LIN {X 0,Y 418.321,Z 60.369,A -85,B 0,C 180,E1 -10243.405,E2 -10243.405} C_VEL
LIN {X 0,Y 418.35,Z 60.367,A -85,B 0,C 180,E1 -10246.999,E2 -10246.999} C_VEL
LIN {X 0,Y 418.344,Z 60.377,A -85,B 0,C 180,E1 -10250.329,E2 -10250.329} C_VEL
LIN {X 0,Y 418.492,Z 60.345,A -85,B 0,C 180,E1 -10253.249,E2 -10253.249} C_VEL
LIN {X 0,Y 418.34,Z 60.372,A -85,B 0,C 180,E1 -10255.181,E2 -10255.181} C_VEL
LIN {X 0,Y 418.544,Z 60.343,A -85,B 0,C 180,E1 -10258.075,E2 -10258.075} C_VEL
LIN {X 0,Y 418.675,Z 60.334,A -85,B 0,C 180,E1 -10260,E2 -10260} C_VEL
LIN {X 0,Y 418.503,Z 60.349,A -85,B 0,C 180,E1 -10262.888,E2 -10262.888} C_VEL
LIN {X 0,Y 418.47,Z 60.356,A -85,B 0,C 180,E1 -10266.618,E2 -10266.618} C_VEL
LIN {X 0,Y 418.342,Z 60.372,A -85,B 0,C 180,E1 -10269.671,E2 -10269.671} C_VEL
LIN {X 0,Y 418.35,Z 60.373,A -85,B 0,C 180,E1 -10273.001,E2 -10273.001} C_VEL
LIN {X 0,Y 418.316,Z 60.378,A -85,B 0,C 180,E1 -10276.735,E2 -10276.735} C_VEL
LIN {X 0,Y 418.273,Z 60.38,A -85,B 0,C 180,E1 -10279.79,E2 -10279.79} C_VEL
LIN {X 0,Y 418.241,Z 60.385,A -85,B 0,C 180,E1 -10282.736,E2 -10282.736} C_VEL
LIN {X 0,Y 418.241,Z 60.384,A -85,B 0,C 180,E1 -10285.906,E2 -10285.906} C_VEL
LIN {X 0,Y 418.263,Z 60.383,A -85,B 0,C 180,E1 -10289.162,E2 -10289.162} C_VEL
LIN {X 0,Y 418.259,Z 60.384,A -85,B 0,C 180,E1 -10292.844,E2 -10292.844} C_VEL
LIN {X 0,Y 418.245,Z 60.388,A -85,B 0,C 180,E1 -10296.237,E2 -10296.237} C_VEL
LIN {X 0,Y 418.23,Z 60.387,A -85,B 0,C 180,E1 -10299.684,E2 -10299.684} C_VEL
LIN {X 0,Y 418.225,Z 60.389,A -85,B 0,C 180,E1 -10302.32,E2 -10302.32} C_VEL
LIN {X 0,Y 418.237,Z 60.387,A -85,B 0,C 180,E1 -10305.108,E2 -10305.108} C_VEL
LIN {X 0,Y 418.235,Z 60.39,A -85,B 0,C 180,E1 -10307.766,E2 -10307.766} C_VEL
LIN {X 0,Y 418.239,Z 60.39,A -85,B 0,C 180,E1 -10311.556,E2 -10311.556} C_VEL
LIN {X 0,Y 418.259,Z 60.389,A -85,B 0,C 180,E1 -10315.159,E2 -10315.159} C_VEL
LIN {X 0,Y 418.265,Z 60.473,A -85,B 0,C 180,E1 -10318.326,E2 -10318.326} C_VEL
LIN {X 0,Y 420.017,Z 68.841,A -85,B 0,C 180,E1 -10320.523,E2 -10320.523} C_VEL
LIN {X 0,Y 423.228,Z 78.508,A -85,B 0,C 180,E1 -10320.878,E2 -10320.878} C_VEL
LIN {X 0,Y 425.271,Z 87.278,A -85,B 0,C 180,E1 -10321.149,E2 -10321.149} C_VEL
LIN {X 0,Y 423.933,Z 175.487,A -85,B 0,C 180,E1 -10322.677,E2 -10322.677} C_VEL
LIN {X 0,Y 423.626,Z 189.114,A -85,B 0,C 180,E1 -10323.123,E2 -10323.123} C_VEL
LIN {X 0,Y 423.181,Z 201.819,A -85,B 0,C 180,E1 -10323.741,E2 -10323.741} C_VEL
LIN {X 0,Y 422.47,Z 213.434,A -85,B 0,C 180,E1 -10324.504,E2 -10324.504} C_VEL
LIN {X 0,Y 421.622,Z 225.198,A -85,B 0,C 180,E1 -10325.503,E2 -10325.503} C_VEL
LIN {X 0,Y 420.814,Z 235.746,A -85,B 0,C 180,E1 -10326.636,E2 -10326.636} C_VEL
LIN {X 0,Y 420.036,Z 245.057,A -85,B 0,C 180,E1 -10327.885,E2 -10327.885} C_VEL
LIN {X 0,Y 419.252,Z 254.097,A -85,B 0,C 180,E1 -10329.389,E2 -10329.389} C_VEL
LIN {X 0,Y 418.577,Z 261.259,A -85,B 0,C 180,E1 -10330.888,E2 -10330.888} C_VEL
LIN {X 0,Y 418.104,Z 266.918,A -85,B 0,C 180,E1 -10332.388,E2 -10332.388} C_VEL
LIN {X 0,Y 417.71,Z 271.445,A -85,B 0,C 180,E1 -10333.932,E2 -10333.932} C_VEL
LIN {X 0,Y 417.433,Z 274.605,A -85,B 0,C 180,E1 -10335.372,E2 -10335.372} C_VEL
LIN {X 0,Y 417.294,Z 276.222,A -85,B 0,C 180,E1 -10336.362,E2 -10336.362} C_VEL
LIN {X 0,Y 417.186,Z 277.725,A -85,B 0,C 180,E1 -10337.709,E2 -10337.709} C_VEL
LIN {X 0,Y 417.089,Z 278.519,A -85,B 0,C 180,E1 -10339.318,E2 -10339.318} C_VEL
LIN {X 0,Y 417.096,Z 278.044,A -85,B 0,C 180,E1 -10341.278,E2 -10341.278} C_VEL
LIN {X 0,Y 417.182,Z 276.739,A -85,B 0,C 180,E1 -10342.584,E2 -10342.584} C_VEL
LIN {X 0,Y 416.579,Z 275.723,A -85,B 0,C 180,E1 -10343.378,E2 -10343.378} C_VEL
LIN {X 0,Y 413.861,Z 273.515,A -85,B 0,C 180,E1 -10344.661,E2 -10344.661} C_VEL
LIN {X 0,Y 411.581,Z 271.313,A -85,B 0,C 180,E1 -10345.676,E2 -10345.676} C_VEL
LIN {X 0,Y 410.648,Z 269.236,A -85,B 0,C 180,E1 -10346.439,E2 -10346.439} C_VEL
LIN {X 0,Y 410.598,Z 268.449,A -85,B 0,C 180,E1 -10346.692,E2 -10346.692} C_VEL
LIN {X 0,Y 410.755,Z 263.792,A -85,B 0,C 180,E1 -10348.039,E2 -10348.039} C_VEL
LIN {X 0,Y 411.262,Z 257.385,A -85,B 0,C 180,E1 -10349.511,E2 -10349.511} C_VEL
LIN {X 0,Y 411.77,Z 249.436,A -85,B 0,C 180,E1 -10350.978,E2 -10350.978} C_VEL
LIN {X 0,Y 412.275,Z 241.341,A -85,B 0,C 180,E1 -10352.198,E2 -10352.198} C_VEL
LIN {X 0,Y 412.997,Z 232.499,A -85,B 0,C 180,E1 -10353.293,E2 -10353.293} C_VEL
LIN {X 0,Y 413.619,Z 222.986,A -85,B 0,C 180,E1 -10354.263,E2 -10354.263} C_VEL
LIN {X 0,Y 414.244,Z 212.762,A -85,B 0,C 180,E1 -10355.11,E2 -10355.11} C_VEL
LIN {X 0,Y 414.76,Z 200.609,A -85,B 0,C 180,E1 -10355.896,E2 -10355.896} C_VEL
LIN {X 0,Y 415.145,Z 187.122,A -85,B 0,C 180,E1 -10356.531,E2 -10356.531} C_VEL
LIN {X 0,Y 415.473,Z 174.29,A -85,B 0,C 180,E1 -10356.922,E2 -10356.922} C_VEL
LIN {X 0,Y 416.386,Z 86.383,A -85,B 0,C 180,E1 -10358.452,E2 -10358.452} C_VEL
LIN {X 0,Y 413.356,Z 71.404,A -85,B 0,C 180,E1 -10358.84,E2 -10358.84} C_VEL
LIN {X 0,Y 412.603,Z 68.628,A -85,B 0,C 180,E1 -10358.936,E2 -10358.936} C_VEL
LIN {X 0,Y 411.29,Z 61.255,A -85,B 0,C 180,E1 -10360.772,E2 -10360.772} C_VEL
LIN {X 0,Y 411.257,Z 61.254,A -85,B 0,C 180,E1 -10363.842,E2 -10363.842} C_VEL
LIN {X 0,Y 411.259,Z 61.256,A -85,B 0,C 180,E1 -10366.889,E2 -10366.889} C_VEL
LIN {X 0,Y 411.232,Z 61.259,A -85,B 0,C 180,E1 -10369.987,E2 -10369.987} C_VEL
LIN {X 0,Y 411.197,Z 61.261,A -85,B 0,C 180,E1 -10373.148,E2 -10373.148} C_VEL
LIN {X 0,Y 411.238,Z 61.26,A -85,B 0,C 180,E1 -10376.381,E2 -10376.381} C_VEL
LIN {X 0,Y 411.202,Z 61.263,A -85,B 0,C 180,E1 -10379.713,E2 -10379.713} C_VEL
LIN {X 0,Y 411.208,Z 61.26,A -85,B 0,C 180,E1 -10383.156,E2 -10383.156} C_VEL
LIN {X 0,Y 411.197,Z 61.261,A -85,B 0,C 180,E1 -10386.553,E2 -10386.553} C_VEL
LIN {X 0,Y 411.221,Z 61.264,A -85,B 0,C 180,E1 -10389.729,E2 -10389.729} C_VEL
LIN {X 0,Y 411.176,Z 61.266,A -85,B 0,C 180,E1 -10393.134,E2 -10393.134} C_VEL
LIN {X 0,Y 411.17,Z 61.266,A -85,B 0,C 180,E1 -10395.881,E2 -10395.881} C_VEL
LIN {X 0,Y 411.166,Z 61.266,A -85,B 0,C 180,E1 -10398.772,E2 -10398.772} C_VEL
LIN {X 0,Y 411.196,Z 61.261,A -85,B 0,C 180,E1 -10402.026,E2 -10402.026} C_VEL
LIN {X 0,Y 411.209,Z 61.26,A -85,B 0,C 180,E1 -10405.667,E2 -10405.667} C_VEL
LIN {X 0,Y 411.193,Z 61.266,A -85,B 0,C 180,E1 -10409.153,E2 -10409.153} C_VEL
LIN {X 0,Y 411.263,Z 61.256,A -85,B 0,C 180,E1 -10412.523,E2 -10412.523} C_VEL
LIN {X 0,Y 411.231,Z 61.257,A -85,B 0,C 180,E1 -10415.785,E2 -10415.785} C_VEL
LIN {X 0,Y 411.201,Z 61.263,A -85,B 0,C 180,E1 -10418.966,E2 -10418.966} C_VEL
LIN {X 0,Y 411.254,Z 61.256,A -85,B 0,C 180,E1 -10422.085,E2 -10422.085} C_VEL
LIN {X 0,Y 411.265,Z 61.253,A -85,B 0,C 180,E1 -10425.148,E2 -10425.148} C_VEL
LIN {X 0,Y 411.288,Z 61.255,A -85,B 0,C 180,E1 -10428.167,E2 -10428.167} C_VEL
LIN {X 0,Y 411.443,Z 61.237,A -85,B 0,C 180,E1 -10432.192,E2 -10432.192} C_VEL
LIN {X 0,Y 411.474,Z 61.233,A -85,B 0,C 180,E1 -10434.118,E2 -10434.118} C_VEL
LIN {X 0,Y 411.514,Z 61.227,A -85,B 0,C 180,E1 -10438.043,E2 -10438.043} C_VEL
LIN {X 0,Y 411.645,Z 61.21,A -85,B 0,C 180,E1 -10440,E2 -10440} C_VEL
LIN {X 0,Y 411.461,Z 61.228,A -85,B 0,C 180,E1 -10442.937,E2 -10442.937} C_VEL
LIN {X 0,Y 411.44,Z 61.235,A -85,B 0,C 180,E1 -10445.883,E2 -10445.883} C_VEL
LIN {X 0,Y 411.324,Z 61.246,A -85,B 0,C 180,E1 -10448.846,E2 -10448.846} C_VEL
LIN {X 0,Y 411.289,Z 61.252,A -85,B 0,C 180,E1 -10451.833,E2 -10451.833} C_VEL
LIN {X 0,Y 411.265,Z 61.254,A -85,B 0,C 180,E1 -10454.853,E2 -10454.853} C_VEL
LIN {X 0,Y 411.25,Z 61.255,A -85,B 0,C 180,E1 -10457.915,E2 -10457.915} C_VEL
LIN {X 0,Y 411.201,Z 61.267,A -85,B 0,C 180,E1 -10461.034,E2 -10461.034} C_VEL
LIN {X 0,Y 411.216,Z 61.259,A -85,B 0,C 180,E1 -10464.216,E2 -10464.216} C_VEL
LIN {X 0,Y 411.212,Z 61.26,A -85,B 0,C 180,E1 -10467.481,E2 -10467.481} C_VEL
LIN {X 0,Y 411.193,Z 61.267,A -85,B 0,C 180,E1 -10470.848,E2 -10470.848} C_VEL
LIN {X 0,Y 411.208,Z 61.263,A -85,B 0,C 180,E1 -10474.334,E2 -10474.334} C_VEL
LIN {X 0,Y 411.195,Z 61.263,A -85,B 0,C 180,E1 -10477.974,E2 -10477.974} C_VEL
LIN {X 0,Y 411.167,Z 61.265,A -85,B 0,C 180,E1 -10481.228,E2 -10481.228} C_VEL
LIN {X 0,Y 411.179,Z 61.267,A -85,B 0,C 180,E1 -10484.49,E2 -10484.49} C_VEL
LIN {X 0,Y 411.175,Z 61.27,A -85,B 0,C 180,E1 -10488.194,E2 -10488.194} C_VEL
LIN {X 0,Y 411.206,Z 61.26,A -85,B 0,C 180,E1 -10490.774,E2 -10490.774} C_VEL
LIN {X 0,Y 411.2,Z 61.262,A -85,B 0,C 180,E1 -10494.471,E2 -10494.471} C_VEL
LIN {X 0,Y 411.21,Z 61.259,A -85,B 0,C 180,E1 -10496.873,E2 -10496.873} C_VEL
LIN {X 0,Y 411.236,Z 61.261,A -85,B 0,C 180,E1 -10500.644,E2 -10500.644} C_VEL
LIN {X 0,Y 411.342,Z 61.377,A -85,B 0,C 180,E1 -10501.802,E2 -10501.802} C_VEL
LIN {X 0,Y 413.981,Z 74.973,A -85,B 0,C 180,E1 -10504.562,E2 -10504.562} C_VEL
LIN {X 0,Y 413.975,Z 79.493,A -85,B 0,C 180,E1 -10505.422,E2 -10505.422} C_VEL
LIN {X 0,Y 412.739,Z 99.028,A -85,B 0,C 180,E1 -10509.048,E2 -10509.048} C_VEL
LIN {X 0,Y 412.207,Z 110.218,A -85,B 0,C 180,E1 -10511.066,E2 -10511.066} C_VEL
LIN {X 0,Y 415.966,Z 140.17,A -85,B 0,C 180,E1 -10511.74,E2 -10511.74} C_VEL
LIN {X 0,Y 415.175,Z 218.857,A -85,B 0,C 180,E1 -10513.117,E2 -10513.117} C_VEL
LIN {X 0,Y 414.652,Z 232.156,A -85,B 0,C 180,E1 -10513.538,E2 -10513.538} C_VEL
LIN {X 0,Y 414.057,Z 244.369,A -85,B 0,C 180,E1 -10514.115,E2 -10514.115} C_VEL
LIN {X 0,Y 413.373,Z 255.873,A -85,B 0,C 180,E1 -10514.847,E2 -10514.847} C_VEL
LIN {X 0,Y 412.617,Z 267.688,A -85,B 0,C 180,E1 -10515.827,E2 -10515.827} C_VEL
LIN {X 0,Y 411.949,Z 278.808,A -85,B 0,C 180,E1 -10516.994,E2 -10516.994} C_VEL
LIN {X 0,Y 411.357,Z 287.857,A -85,B 0,C 180,E1 -10518.169,E2 -10518.169} C_VEL
LIN {X 0,Y 410.7,Z 297.04,A -85,B 0,C 180,E1 -10519.649,E2 -10519.649} C_VEL
LIN {X 0,Y 410.339,Z 304.446,A -85,B 0,C 180,E1 -10521.133,E2 -10521.133} C_VEL
LIN {X 0,Y 410.157,Z 310.38,A -85,B 0,C 180,E1 -10522.616,E2 -10522.616} C_VEL
LIN {X 0,Y 409.977,Z 315.039,A -85,B 0,C 180,E1 -10524.096,E2 -10524.096} C_VEL
LIN {X 0,Y 410.018,Z 318.584,A -85,B 0,C 180,E1 -10525.576,E2 -10525.576} C_VEL
LIN {X 0,Y 410.084,Z 321.104,A -85,B 0,C 180,E1 -10527.053,E2 -10527.053} C_VEL
LIN {X 0,Y 410.064,Z 322.26,A -85,B 0,C 180,E1 -10528.036,E2 -10528.036} C_VEL
LIN {X 0,Y 410.037,Z 323.304,A -85,B 0,C 180,E1 -10530,E2 -10530} C_VEL
LIN {X 0,Y 410.012,Z 323.241,A -85,B 0,C 180,E1 -10530.982,E2 -10530.982} C_VEL
LIN {X 0,Y 410.046,Z 322.783,A -85,B 0,C 180,E1 -10531.964,E2 -10531.964} C_VEL
LIN {X 0,Y 410.026,Z 321.885,A -85,B 0,C 180,E1 -10532.947,E2 -10532.947} C_VEL
LIN {X 0,Y 410.003,Z 318.893,A -85,B 0,C 180,E1 -10534.917,E2 -10534.917} C_VEL
LIN {X 0,Y 409.995,Z 315.492,A -85,B 0,C 180,E1 -10536.397,E2 -10536.397} C_VEL
LIN {X 0,Y 410.228,Z 311.027,A -85,B 0,C 180,E1 -10537.877,E2 -10537.877} C_VEL
LIN {X 0,Y 410.613,Z 304.302,A -85,B 0,C 180,E1 -10539.606,E2 -10539.606} C_VEL
LIN {X 0,Y 411.138,Z 296.984,A -85,B 0,C 180,E1 -10541.087,E2 -10541.087} C_VEL
LIN {X 0,Y 411.853,Z 289.569,A -85,B 0,C 180,E1 -10542.316,E2 -10542.316} C_VEL
LIN {X 0,Y 412.531,Z 280.611,A -85,B 0,C 180,E1 -10543.547,E2 -10543.547} C_VEL
LIN {X 0,Y 413.387,Z 270.909,A -85,B 0,C 180,E1 -10544.636,E2 -10544.636} C_VEL
LIN {X 0,Y 414.351,Z 260.002,A -85,B 0,C 180,E1 -10545.62,E2 -10545.62} C_VEL
LIN {X 0,Y 415.226,Z 247.925,A -85,B 0,C 180,E1 -10546.47,E2 -10546.47} C_VEL
LIN {X 0,Y 416.093,Z 235.332,A -85,B 0,C 180,E1 -10547.129,E2 -10547.129} C_VEL
LIN {X 0,Y 416.772,Z 223.06,A -85,B 0,C 180,E1 -10547.575,E2 -10547.575} C_VEL
LIN {X 0,Y 417.078,Z 208.583,A -85,B 0,C 180,E1 -10547.892,E2 -10547.892} C_VEL
LIN {X 0,Y 417.896,Z 139.431,A -85,B 0,C 180,E1 -10549.103,E2 -10549.103} C_VEL
LIN {X 0,Y 414.917,Z 119.679,A -85,B 0,C 180,E1 -10549.627,E2 -10549.627} C_VEL
LIN {X 0,Y 413.071,Z 109.315,A -85,B 0,C 180,E1 -10549.946,E2 -10549.946} C_VEL
LIN {X 0,Y 414.405,Z 89.718,A -85,B 0,C 180,E1 -10553.68,E2 -10553.68} C_VEL
LIN {X 0,Y 415.149,Z 79.901,A -85,B 0,C 180,E1 -10555.575,E2 -10555.575} C_VEL
LIN {X 0,Y 413.376,Z 70.403,A -85,B 0,C 180,E1 -10557.607,E2 -10557.607} C_VEL
LIN {X 0,Y 411.225,Z 61.262,A -85,B 0,C 180,E1 -10559.682,E2 -10559.682} C_VEL
LIN {X 0,Y 411.209,Z 61.263,A -85,B 0,C 180,E1 -10563.156,E2 -10563.156} C_VEL
LIN {X 0,Y 411.195,Z 61.264,A -85,B 0,C 180,E1 -10566.553,E2 -10566.553} C_VEL
LIN {X 0,Y 411.215,Z 61.254,A -85,B 0,C 180,E1 -10569.728,E2 -10569.728} C_VEL
LIN {X 0,Y 411.176,Z 61.263,A -85,B 0,C 180,E1 -10573.134,E2 -10573.134} C_VEL
LIN {X 0,Y 411.17,Z 61.266,A -85,B 0,C 180,E1 -10575.881,E2 -10575.881} C_VEL
LIN {X 0,Y 411.166,Z 61.263,A -85,B 0,C 180,E1 -10578.772,E2 -10578.772} C_VEL
LIN {X 0,Y 411.195,Z 61.26,A -85,B 0,C 180,E1 -10582.026,E2 -10582.026} C_VEL
LIN {X 0,Y 411.207,Z 61.258,A -85,B 0,C 180,E1 -10585.666,E2 -10585.666} C_VEL
LIN {X 0,Y 411.193,Z 61.264,A -85,B 0,C 180,E1 -10589.152,E2 -10589.152} C_VEL
LIN {X 0,Y 411.262,Z 61.256,A -85,B 0,C 180,E1 -10592.522,E2 -10592.522} C_VEL
LIN {X 0,Y 411.23,Z 61.258,A -85,B 0,C 180,E1 -10595.785,E2 -10595.785} C_VEL
LIN {X 0,Y 411.2,Z 61.262,A -85,B 0,C 180,E1 -10598.966,E2 -10598.966} C_VEL
LIN {X 0,Y 411.256,Z 61.255,A -85,B 0,C 180,E1 -10602.085,E2 -10602.085} C_VEL
LIN {X 0,Y 411.264,Z 61.254,A -85,B 0,C 180,E1 -10605.147,E2 -10605.147} C_VEL
LIN {X 0,Y 411.288,Z 61.247,A -85,B 0,C 180,E1 -10608.167,E2 -10608.167} C_VEL
LIN {X 0,Y 411.444,Z 61.229,A -85,B 0,C 180,E1 -10612.189,E2 -10612.189} C_VEL
LIN {X 0,Y 411.476,Z 61.226,A -85,B 0,C 180,E1 -10614.118,E2 -10614.118} C_VEL
LIN {X 0,Y 411.513,Z 61.219,A -85,B 0,C 180,E1 -10618.042,E2 -10618.042} C_VEL
LIN {X 0,Y 411.644,Z 61.21,A -85,B 0,C 180,E1 -10620,E2 -10620} C_VEL
LIN {X 0,Y 411.46,Z 61.226,A -85,B 0,C 180,E1 -10622.937,E2 -10622.937} C_VEL
LIN {X 0,Y 411.433,Z 61.233,A -85,B 0,C 180,E1 -10626.618,E2 -10626.618} C_VEL
LIN {X 0,Y 411.322,Z 61.241,A -85,B 0,C 180,E1 -10628.846,E2 -10628.846} C_VEL
LIN {X 0,Y 411.287,Z 61.252,A -85,B 0,C 180,E1 -10631.833,E2 -10631.833} C_VEL
LIN {X 0,Y 411.264,Z 61.25,A -85,B 0,C 180,E1 -10634.852,E2 -10634.852} C_VEL
LIN {X 0,Y 411.249,Z 61.252,A -85,B 0,C 180,E1 -10637.915,E2 -10637.915} C_VEL
LIN {X 0,Y 411.199,Z 61.267,A -85,B 0,C 180,E1 -10641.034,E2 -10641.034} C_VEL
LIN {X 0,Y 411.221,Z 61.258,A -85,B 0,C 180,E1 -10644.216,E2 -10644.216} C_VEL
LIN {X 0,Y 411.21,Z 61.258,A -85,B 0,C 180,E1 -10647.481,E2 -10647.481} C_VEL
LIN {X 0,Y 411.191,Z 61.264,A -85,B 0,C 180,E1 -10650.847,E2 -10650.847} C_VEL
LIN {X 0,Y 411.206,Z 61.262,A -85,B 0,C 180,E1 -10654.333,E2 -10654.333} C_VEL
LIN {X 0,Y 411.188,Z 61.265,A -85,B 0,C 180,E1 -10657.974,E2 -10657.974} C_VEL
LIN {X 0,Y 411.159,Z 61.258,A -85,B 0,C 180,E1 -10661.227,E2 -10661.227} C_VEL
LIN {X 0,Y 411.177,Z 61.269,A -85,B 0,C 180,E1 -10664.49,E2 -10664.49} C_VEL
LIN {X 0,Y 411.173,Z 61.269,A -85,B 0,C 180,E1 -10668.194,E2 -10668.194} C_VEL
LIN {X 0,Y 411.184,Z 61.265,A -85,B 0,C 180,E1 -10670.772,E2 -10670.772} C_VEL
LIN {X 0,Y 411.197,Z 61.266,A -85,B 0,C 180,E1 -10674.471,E2 -10674.471} C_VEL
LIN {X 0,Y 411.241,Z 61.335,A -85,B 0,C 180,E1 -10678.009,E2 -10678.009} C_VEL
LIN {X 0,Y 412.934,Z 69.455,A -85,B 0,C 180,E1 -10680.121,E2 -10680.121} C_VEL
LIN {X 0,Y 416.644,Z 79.822,A -85,B 0,C 180,E1 -10680.53,E2 -10680.53} C_VEL
LIN {X 0,Y 418.674,Z 88.026,A -85,B 0,C 180,E1 -10680.796,E2 -10680.796} C_VEL
LIN {X 0,Y 417.293,Z 175.806,A -85,B 0,C 180,E1 -10682.341,E2 -10682.341} C_VEL
LIN {X 0,Y 416.956,Z 189.447,A -85,B 0,C 180,E1 -10682.793,E2 -10682.793} C_VEL
LIN {X 0,Y 416.487,Z 202.219,A -85,B 0,C 180,E1 -10683.425,E2 -10683.425} C_VEL
LIN {X 0,Y 415.759,Z 213.791,A -85,B 0,C 180,E1 -10684.197,E2 -10684.197} C_VEL
LIN {X 0,Y 414.858,Z 225.555,A -85,B 0,C 180,E1 -10685.211,E2 -10685.211} C_VEL
LIN {X 0,Y 414.039,Z 235.627,A -85,B 0,C 180,E1 -10686.302,E2 -10686.302} C_VEL
LIN {X 0,Y 413.277,Z 244.592,A -85,B 0,C 180,E1 -10687.504,E2 -10687.504} C_VEL
LIN {X 0,Y 412.4,Z 253.773,A -85,B 0,C 180,E1 -10689.03,E2 -10689.03} C_VEL
LIN {X 0,Y 411.682,Z 261.104,A -85,B 0,C 180,E1 -10690.555,E2 -10690.555} C_VEL
LIN {X 0,Y 411.146,Z 266.882,A -85,B 0,C 180,E1 -10692.08,E2 -10692.08} C_VEL
LIN {X 0,Y 410.821,Z 270.686,A -85,B 0,C 180,E1 -10693.336,E2 -10693.336} C_VEL
LIN {X 0,Y 410.404,Z 274.759,A -85,B 0,C 180,E1 -10695.116,E2 -10695.116} C_VEL
LIN {X 0,Y 410.266,Z 276.419,A -85,B 0,C 180,E1 -10696.124,E2 -10696.124} C_VEL
LIN {X 0,Y 410.131,Z 278.108,A -85,B 0,C 180,E1 -10697.621,E2 -10697.621} C_VEL
LIN {X 0,Y 410.021,Z 278.885,A -85,B 0,C 180,E1 -10699.132,E2 -10699.132} C_VEL
LIN {X 0,Y 410.005,Z 278.498,A -85,B 0,C 180,E1 -10701.125,E2 -10701.125} C_VEL
LIN {X 0,Y 410.102,Z 277.101,A -85,B 0,C 180,E1 -10702.603,E2 -10702.603} C_VEL
LIN {X 0,Y 410.282,Z 274.842,A -85,B 0,C 180,E1 -10704.101,E2 -10704.101} C_VEL
LIN {X 0,Y 410.374,Z 271.592,A -85,B 0,C 180,E1 -10705.58,E2 -10705.58} C_VEL
LIN {X 0,Y 410.598,Z 268.449,A -85,B 0,C 180,E1 -10706.692,E2 -10706.692} C_VEL
LIN {X 0,Y 410.053,Z 266.051,A -85,B 0,C 180,E1 -10707.439,E2 -10707.439} C_VEL
LIN {X 0,Y 406.327,Z 259.878,A -85,B 0,C 180,E1 -10709.108,E2 -10709.108} C_VEL
LIN {X 0,Y 404.688,Z 255.733,A -85,B 0,C 180,E1 -10710.035,E2 -10710.035} C_VEL
LIN {X 0,Y 404.529,Z 253.406,A -85,B 0,C 180,E1 -10710.487,E2 -10710.487} C_VEL
LIN {X 0,Y 405.115,Z 244.366,A -85,B 0,C 180,E1 -10711.988,E2 -10711.988} C_VEL
LIN {X 0,Y 405.793,Z 235.038,A -85,B 0,C 180,E1 -10713.227,E2 -10713.227} C_VEL
LIN {X 0,Y 406.581,Z 224.672,A -85,B 0,C 180,E1 -10714.337,E2 -10714.337} C_VEL
LIN {X 0,Y 407.331,Z 213.166,A -85,B 0,C 180,E1 -10715.321,E2 -10715.321} C_VEL
LIN {X 0,Y 407.871,Z 201.02,A -85,B 0,C 180,E1 -10716.12,E2 -10716.12} C_VEL
LIN {X 0,Y 408.271,Z 187.541,A -85,B 0,C 180,E1 -10716.766,E2 -10716.766} C_VEL
LIN {X 0,Y 408.608,Z 174.746,A -85,B 0,C 180,E1 -10717.164,E2 -10717.164} C_VEL
LIN {X 0,Y 409.625,Z 87.553,A -85,B 0,C 180,E1 -10718.703,E2 -10718.703} C_VEL
LIN {X 0,Y 406.631,Z 72.984,A -85,B 0,C 180,E1 -10719.09,E2 -10719.09} C_VEL
LIN {X 0,Y 405.499,Z 69.013,A -85,B 0,C 180,E1 -10719.22,E2 -10719.22} C_VEL
LIN {X 0,Y 404.256,Z 62.129,A -85,B 0,C 180,E1 -10720.962,E2 -10720.962} C_VEL
LIN {X 0,Y 404.212,Z 62.133,A -85,B 0,C 180,E1 -10724.088,E2 -10724.088} C_VEL
LIN {X 0,Y 404.205,Z 62.132,A -85,B 0,C 180,E1 -10727.193,E2 -10727.193} C_VEL
LIN {X 0,Y 404.188,Z 62.141,A -85,B 0,C 180,E1 -10730.351,E2 -10730.351} C_VEL
LIN {X 0,Y 404.165,Z 62.138,A -85,B 0,C 180,E1 -10733.575,E2 -10733.575} C_VEL
LIN {X 0,Y 404.185,Z 62.137,A -85,B 0,C 180,E1 -10735.767,E2 -10735.767} C_VEL
LIN {X 0,Y 404.197,Z 62.139,A -85,B 0,C 180,E1 -10738,E2 -10738} C_VEL
LIN {X 0,Y 404.141,Z 62.142,A -85,B 0,C 180,E1 -10741.558,E2 -10741.558} C_VEL
LIN {X 0,Y 404.188,Z 62.134,A -85,B 0,C 180,E1 -10745.016,E2 -10745.016} C_VEL
LIN {X 0,Y 404.161,Z 62.137,A -85,B 0,C 180,E1 -10748.757,E2 -10748.757} C_VEL
LIN {X 0,Y 404.126,Z 62.149,A -85,B 0,C 180,E1 -10751.6,E2 -10751.6} C_VEL
LIN {X 0,Y 404.148,Z 62.139,A -85,B 0,C 180,E1 -10754.522,E2 -10754.522} C_VEL
LIN {X 0,Y 404.139,Z 62.146,A -85,B 0,C 180,E1 -10757.296,E2 -10757.296} C_VEL
LIN {X 0,Y 404.171,Z 62.137,A -85,B 0,C 180,E1 -10759.956,E2 -10759.956} C_VEL
LIN {X 0,Y 404.139,Z 62.146,A -85,B 0,C 180,E1 -10763.125,E2 -10763.125} C_VEL
LIN {X 0,Y 404.148,Z 62.139,A -85,B 0,C 180,E1 -10766.188,E2 -10766.188} C_VEL
LIN {X 0,Y 404.149,Z 62.139,A -85,B 0,C 180,E1 -10769.715,E2 -10769.715} C_VEL
LIN {X 0,Y 404.199,Z 62.136,A -85,B 0,C 180,E1 -10773.123,E2 -10773.123} C_VEL
LIN {X 0,Y 404.181,Z 62.136,A -85,B 0,C 180,E1 -10775.335,E2 -10775.335} C_VEL
LIN {X 0,Y 404.164,Z 62.143,A -85,B 0,C 180,E1 -10778.582,E2 -10778.582} C_VEL
LIN {X 0,Y 404.212,Z 62.131,A -85,B 0,C 180,E1 -10781.762,E2 -10781.762} C_VEL
LIN {X 0,Y 404.211,Z 62.133,A -85,B 0,C 180,E1 -10784.882,E2 -10784.882} C_VEL
LIN {X 0,Y 404.261,Z 62.128,A -85,B 0,C 180,E1 -10787.959,E2 -10787.959} C_VEL
LIN {X 0,Y 404.408,Z 62.113,A -85,B 0,C 180,E1 -10792.131,E2 -10792.131} C_VEL
LIN {X 0,Y 404.421,Z 62.111,A -85,B 0,C 180,E1 -10794.015,E2 -10794.015} C_VEL
LIN {X 0,Y 404.483,Z 62.103,A -85,B 0,C 180,E1 -10798.009,E2 -10798.009} C_VEL
LIN {X 0,Y 404.615,Z 62.086,A -85,B 0,C 180,E1 -10800,E2 -10800} C_VEL
LIN {X 0,Y 404.419,Z 62.105,A -85,B 0,C 180,E1 -10802.989,E2 -10802.989} C_VEL
LIN {X 0,Y 404.387,Z 62.112,A -85,B 0,C 180,E1 -10805.986,E2 -10805.986} C_VEL
LIN {X 0,Y 404.271,Z 62.125,A -85,B 0,C 180,E1 -10809.002,E2 -10809.002} C_VEL
LIN {X 0,Y 404.261,Z 62.126,A -85,B 0,C 180,E1 -10812.042,E2 -10812.042} C_VEL
LIN {X 0,Y 404.211,Z 62.136,A -85,B 0,C 180,E1 -10815.118,E2 -10815.118} C_VEL
LIN {X 0,Y 404.209,Z 62.131,A -85,B 0,C 180,E1 -10818.238,E2 -10818.238} C_VEL
LIN {X 0,Y 404.143,Z 62.143,A -85,B 0,C 180,E1 -10821.419,E2 -10821.419} C_VEL
LIN {X 0,Y 404.168,Z 62.14,A -85,B 0,C 180,E1 -10824.666,E2 -10824.666} C_VEL
LIN {X 0,Y 404.172,Z 62.136,A -85,B 0,C 180,E1 -10828.002,E2 -10828.002} C_VEL
LIN {X 0,Y 404.143,Z 62.14,A -85,B 0,C 180,E1 -10831.558,E2 -10831.558} C_VEL
LIN {X 0,Y 404.187,Z 62.136,A -85,B 0,C 180,E1 -10835.016,E2 -10835.016} C_VEL
LIN {X 0,Y 404.154,Z 62.142,A -85,B 0,C 180,E1 -10838.757,E2 -10838.757} C_VEL
LIN {X 0,Y 404.126,Z 62.142,A -85,B 0,C 180,E1 -10841.6,E2 -10841.6} C_VEL
LIN {X 0,Y 404.148,Z 62.143,A -85,B 0,C 180,E1 -10844.522,E2 -10844.522} C_VEL
LIN {X 0,Y 404.136,Z 62.141,A -85,B 0,C 180,E1 -10847.295,E2 -10847.295} C_VEL
LIN {X 0,Y 404.137,Z 62.146,A -85,B 0,C 180,E1 -10849.951,E2 -10849.951} C_VEL
LIN {X 0,Y 404.137,Z 62.14,A -85,B 0,C 180,E1 -10853.125,E2 -10853.125} C_VEL
LIN {X 0,Y 404.147,Z 62.142,A -85,B 0,C 180,E1 -10856.188,E2 -10856.188} C_VEL
LIN {X 0,Y 404.149,Z 62.146,A -85,B 0,C 180,E1 -10859.715,E2 -10859.715} C_VEL
LIN {X 0,Y 404.277,Z 62.27,A -85,B 0,C 180,E1 -10861.582,E2 -10861.582} C_VEL
LIN {X 0,Y 406.96,Z 75.991,A -85,B 0,C 180,E1 -10864.422,E2 -10864.422} C_VEL
LIN {X 0,Y 407.03,Z 80.23,A -85,B 0,C 180,E1 -10865.246,E2 -10865.246} C_VEL
LIN {X 0,Y 405.746,Z 99.417,A -85,B 0,C 180,E1 -10868.871,E2 -10868.871} C_VEL
LIN {X 0,Y 405.251,Z 109.671,A -85,B 0,C 180,E1 -10870.778,E2 -10870.778} C_VEL
LIN {X 0,Y 409.126,Z 139.835,A -85,B 0,C 180,E1 -10871.474,E2 -10871.474} C_VEL
LIN {X 0,Y 408.291,Z 219.024,A -85,B 0,C 180,E1 -10872.888,E2 -10872.888} C_VEL
LIN {X 0,Y 407.668,Z 232.897,A -85,B 0,C 180,E1 -10873.345,E2 -10873.345} C_VEL
LIN {X 0,Y 407.096,Z 245.367,A -85,B 0,C 180,E1 -10873.965,E2 -10873.965} C_VEL
LIN {X 0,Y 406.366,Z 256.491,A -85,B 0,C 180,E1 -10874.707,E2 -10874.707} C_VEL
LIN {X 0,Y 405.589,Z 268.116,A -85,B 0,C 180,E1 -10875.704,E2 -10875.704} C_VEL
LIN {X 0,Y 404.968,Z 278.258,A -85,B 0,C 180,E1 -10876.794,E2 -10876.794} C_VEL
LIN {X 0,Y 404.334,Z 287.149,A -85,B 0,C 180,E1 -10877.961,E2 -10877.961} C_VEL
LIN {X 0,Y 403.685,Z 296.404,A -85,B 0,C 180,E1 -10879.467,E2 -10879.467} C_VEL
LIN {X 0,Y 403.288,Z 303.855,A -85,B 0,C 180,E1 -10880.976,E2 -10880.976} C_VEL
LIN {X 0,Y 403.066,Z 309.828,A -85,B 0,C 180,E1 -10882.486,E2 -10882.486} C_VEL
LIN {X 0,Y 402.899,Z 314.526,A -85,B 0,C 180,E1 -10883.992,E2 -10883.992} C_VEL
LIN {X 0,Y 402.947,Z 318.104,A -85,B 0,C 180,E1 -10885.498,E2 -10885.498} C_VEL
LIN {X 0,Y 402.983,Z 320.653,A -85,B 0,C 180,E1 -10887.001,E2 -10887.001} C_VEL
LIN {X 0,Y 402.993,Z 321.837,A -85,B 0,C 180,E1 -10888.001,E2 -10888.001} C_VEL
LIN {X 0,Y 402.959,Z 322.571,A -85,B 0,C 180,E1 -10889.001,E2 -10889.001} C_VEL
LIN {X 0,Y 402.956,Z 322.912,A -85,B 0,C 180,E1 -10890,E2 -10890} C_VEL
LIN {X 0,Y 402.974,Z 322.427,A -85,B 0,C 180,E1 -10891.999,E2 -10891.999} C_VEL
LIN {X 0,Y 402.924,Z 321.549,A -85,B 0,C 180,E1 -10892.999,E2 -10892.999} C_VEL
LIN {X 0,Y 402.909,Z 318.586,A -85,B 0,C 180,E1 -10895.003,E2 -10895.003} C_VEL
LIN {X 0,Y 402.922,Z 315.217,A -85,B 0,C 180,E1 -10896.509,E2 -10896.509} C_VEL
LIN {X 0,Y 403.17,Z 310.788,A -85,B 0,C 180,E1 -10898.016,E2 -10898.016} C_VEL
LIN {X 0,Y 403.496,Z 305.176,A -85,B 0,C 180,E1 -10899.524,E2 -10899.524} C_VEL
LIN {X 0,Y 404.003,Z 298.197,A -85,B 0,C 180,E1 -10901.032,E2 -10901.032} C_VEL
LIN {X 0,Y 404.894,Z 289.486,A -85,B 0,C 180,E1 -10902.531,E2 -10902.531} C_VEL
LIN {X 0,Y 405.664,Z 279.998,A -85,B 0,C 180,E1 -10903.859,E2 -10903.859} C_VEL
LIN {X 0,Y 406.635,Z 269.669,A -85,B 0,C 180,E1 -10905.026,E2 -10905.026} C_VEL
LIN {X 0,Y 407.634,Z 258.647,A -85,B 0,C 180,E1 -10906.013,E2 -10906.013} C_VEL
LIN {X 0,Y 408.441,Z 248.309,A -85,B 0,C 180,E1 -10906.751,E2 -10906.751} C_VEL
LIN {X 0,Y 409.344,Z 235.957,A -85,B 0,C 180,E1 -10907.421,E2 -10907.421} C_VEL
LIN {X 0,Y 410.083,Z 223.26,A -85,B 0,C 180,E1 -10907.903,E2 -10907.903} C_VEL
LIN {X 0,Y 410.437,Z 208.997,A -85,B 0,C 180,E1 -10908.228,E2 -10908.228} C_VEL
LIN {X 0,Y 411.262,Z 139.533,A -85,B 0,C 180,E1 -10909.466,E2 -10909.466} C_VEL
LIN {X 0,Y 407.373,Z 115.504,A -85,B 0,C 180,E1 -10910.138,E2 -10910.138} C_VEL
LIN {X 0,Y 406.2,Z 109.031,A -85,B 0,C 180,E1 -10910.332,E2 -10910.332} C_VEL
LIN {X 0,Y 407.645,Z 89.572,A -85,B 0,C 180,E1 -10914.107,E2 -10914.107} C_VEL
LIN {X 0,Y 408.3,Z 81.425,A -85,B 0,C 180,E1 -10915.71,E2 -10915.71} C_VEL
LIN {X 0,Y 406.212,Z 70.646,A -85,B 0,C 180,E1 -10918.07,E2 -10918.07} C_VEL
LIN {X 0,Y 404.192,Z 62.139,A -85,B 0,C 180,E1 -10920.046,E2 -10920.046} C_VEL
LIN {X 0,Y 404.147,Z 62.144,A -85,B 0,C 180,E1 -10923.812,E2 -10923.812} C_VEL
LIN {X 0,Y 404.139,Z 62.142,A -85,B 0,C 180,E1 -10926.875,E2 -10926.875} C_VEL
LIN {X 0,Y 404.15,Z 62.136,A -85,B 0,C 180,E1 -10930.08,E2 -10930.08} C_VEL
LIN {X 0,Y 404.156,Z 62.137,A -85,B 0,C 180,E1 -10933.084,E2 -10933.084} C_VEL
LIN {X 0,Y 404.151,Z 62.14,A -85,B 0,C 180,E1 -10935.926,E2 -10935.926} C_VEL
LIN {X 0,Y 404.121,Z 62.141,A -85,B 0,C 180,E1 -10938.635,E2 -10938.635} C_VEL
LIN {X 0,Y 404.153,Z 62.142,A -85,B 0,C 180,E1 -10941.493,E2 -10941.493} C_VEL
LIN {X 0,Y 404.187,Z 62.137,A -85,B 0,C 180,E1 -10944.984,E2 -10944.984} C_VEL
LIN {X 0,Y 404.145,Z 62.142,A -85,B 0,C 180,E1 -10948.554,E2 -10948.554} C_VEL
LIN {X 0,Y 404.199,Z 62.134,A -85,B 0,C 180,E1 -10952,E2 -10952} C_VEL
LIN {X 0,Y 404.181,Z 62.138,A -85,B 0,C 180,E1 -10955.334,E2 -10955.334} C_VEL
LIN {X 0,Y 404.142,Z 62.139,A -85,B 0,C 180,E1 -10958.581,E2 -10958.581} C_VEL
LIN {X 0,Y 404.214,Z 62.131,A -85,B 0,C 180,E1 -10961.762,E2 -10961.762} C_VEL
LIN {X 0,Y 404.21,Z 62.134,A -85,B 0,C 180,E1 -10964.882,E2 -10964.882} C_VEL
LIN {X 0,Y 404.26,Z 62.122,A -85,B 0,C 180,E1 -10967.958,E2 -10967.958} C_VEL
LIN {X 0,Y 404.409,Z 62.106,A -85,B 0,C 180,E1 -10972.129,E2 -10972.129} C_VEL
LIN {X 0,Y 404.424,Z 62.103,A -85,B 0,C 180,E1 -10974.015,E2 -10974.015} C_VEL
LIN {X 0,Y 404.482,Z 62.095,A -85,B 0,C 180,E1 -10978.008,E2 -10978.008} C_VEL
LIN {X 0,Y 404.614,Z 62.085,A -85,B 0,C 180,E1 -10980,E2 -10980} C_VEL
LIN {X 0,Y 404.418,Z 62.103,A -85,B 0,C 180,E1 -10982.988,E2 -10982.988} C_VEL
LIN {X 0,Y 404.383,Z 62.111,A -85,B 0,C 180,E1 -10986.617,E2 -10986.617} C_VEL
LIN {X 0,Y 404.269,Z 62.12,A -85,B 0,C 180,E1 -10989.001,E2 -10989.001} C_VEL
LIN {X 0,Y 404.26,Z 62.126,A -85,B 0,C 180,E1 -10992.041,E2 -10992.041} C_VEL
LIN {X 0,Y 404.21,Z 62.132,A -85,B 0,C 180,E1 -10995.118,E2 -10995.118} C_VEL
LIN {X 0,Y 404.207,Z 62.129,A -85,B 0,C 180,E1 -10998.238,E2 -10998.238} C_VEL
LIN {X 0,Y 404.142,Z 62.142,A -85,B 0,C 180,E1 -11001.419,E2 -11001.419} C_VEL
LIN {X 0,Y 404.175,Z 62.139,A -85,B 0,C 180,E1 -11004.666,E2 -11004.666} C_VEL
LIN {X 0,Y 404.17,Z 62.136,A -85,B 0,C 180,E1 -11008.001,E2 -11008.001} C_VEL
LIN {X 0,Y 404.141,Z 62.14,A -85,B 0,C 180,E1 -11011.558,E2 -11011.558} C_VEL
LIN {X 0,Y 404.185,Z 62.137,A -85,B 0,C 180,E1 -11015.016,E2 -11015.016} C_VEL
LIN {X 0,Y 404.144,Z 62.142,A -85,B 0,C 180,E1 -11018.758,E2 -11018.758} C_VEL
LIN {X 0,Y 404.118,Z 62.136,A -85,B 0,C 180,E1 -11021.599,E2 -11021.599} C_VEL
LIN {X 0,Y 404.146,Z 62.144,A -85,B 0,C 180,E1 -11024.522,E2 -11024.522} C_VEL
LIN {X 0,Y 404.134,Z 62.145,A -85,B 0,C 180,E1 -11027.295,E2 -11027.295} C_VEL
LIN {X 0,Y 404.133,Z 62.147,A -85,B 0,C 180,E1 -11029.951,E2 -11029.951} C_VEL
LIN {X 0,Y 404.135,Z 62.146,A -85,B 0,C 180,E1 -11033.125,E2 -11033.125} C_VEL
LIN {X 0,Y 404.145,Z 62.145,A -85,B 0,C 180,E1 -11036.188,E2 -11036.188} C_VEL
LIN {X 0,Y 404.179,Z 62.227,A -85,B 0,C 180,E1 -11037.678,E2 -11037.678} C_VEL
LIN {X 0,Y 405.733,Z 69.688,A -85,B 0,C 180,E1 -11039.689,E2 -11039.689} C_VEL
LIN {X 0,Y 410.05,Z 80.961,A -85,B 0,C 180,E1 -11040.164,E2 -11040.164} C_VEL
LIN {X 0,Y 412.084,Z 88.998,A -85,B 0,C 180,E1 -11040.435,E2 -11040.435} C_VEL
LIN {X 0,Y 410.667,Z 176.173,A -85,B 0,C 180,E1 -11041.994,E2 -11041.994} C_VEL
LIN {X 0,Y 410.327,Z 189.825,A -85,B 0,C 180,E1 -11042.455,E2 -11042.455} C_VEL
LIN {X 0,Y 409.824,Z 202.543,A -85,B 0,C 180,E1 -11043.093,E2 -11043.093} C_VEL
LIN {X 0,Y 409.045,Z 214.162,A -85,B 0,C 180,E1 -11043.878,E2 -11043.878} C_VEL
LIN {X 0,Y 408.098,Z 225.929,A -85,B 0,C 180,E1 -11044.908,E2 -11044.908} C_VEL
LIN {X 0,Y 407.269,Z 235.502,A -85,B 0,C 180,E1 -11045.957,E2 -11045.957} C_VEL
LIN {X 0,Y 406.504,Z 244.102,A -85,B 0,C 180,E1 -11047.108,E2 -11047.108} C_VEL
LIN {X 0,Y 405.676,Z 252.071,A -85,B 0,C 180,E1 -11048.399,E2 -11048.399} C_VEL
LIN {X 0,Y 404.894,Z 259.78,A -85,B 0,C 180,E1 -11049.952,E2 -11049.952} C_VEL
LIN {X 0,Y 404.19,Z 266.838,A -85,B 0,C 180,E1 -11051.761,E2 -11051.761} C_VEL
LIN {X 0,Y 403.788,Z 271.134,A -85,B 0,C 180,E1 -11053.193,E2 -11053.193} C_VEL
LIN {X 0,Y 403.386,Z 274.913,A -85,B 0,C 180,E1 -11054.85,E2 -11054.85} C_VEL
LIN {X 0,Y 403.225,Z 276.62,A -85,B 0,C 180,E1 -11055.876,E2 -11055.876} C_VEL
LIN {X 0,Y 403.067,Z 278.497,A -85,B 0,C 180,E1 -11057.536,E2 -11057.536} C_VEL
LIN {X 0,Y 402.963,Z 279.251,A -85,B 0,C 180,E1 -11058.939,E2 -11058.939} C_VEL
LIN {X 0,Y 402.902,Z 278.947,A -85,B 0,C 180,E1 -11060.968,E2 -11060.968} C_VEL
LIN {X 0,Y 402.98,Z 278.213,A -85,B 0,C 180,E1 -11061.98,E2 -11061.98} C_VEL
LIN {X 0,Y 403.154,Z 276.238,A -85,B 0,C 180,E1 -11063.543,E2 -11063.543} C_VEL
LIN {X 0,Y 403.27,Z 272.294,A -85,B 0,C 180,E1 -11065.502,E2 -11065.502} C_VEL
LIN {X 0,Y 403.588,Z 268.064,A -85,B 0,C 180,E1 -11067.005,E2 -11067.005} C_VEL
LIN {X 0,Y 403.876,Z 261.689,A -85,B 0,C 180,E1 -11068.754,E2 -11068.754} C_VEL
LIN {X 0,Y 404.453,Z 254.688,A -85,B 0,C 180,E1 -11070.249,E2 -11070.249} C_VEL
LIN {X 0,Y 404.529,Z 253.406,A -85,B 0,C 180,E1 -11070.487,E2 -11070.487} C_VEL
LIN {X 0,Y 404.119,Z 249.817,A -85,B 0,C 180,E1 -11071.145,E2 -11071.145} C_VEL
LIN {X 0,Y 401.769,Z 243.676,A -85,B 0,C 180,E1 -11072.194,E2 -11072.194} C_VEL
LIN {X 0,Y 399.471,Z 237.013,A -85,B 0,C 180,E1 -11073.188,E2 -11073.188} C_VEL
LIN {X 0,Y 399.14,Z 232.544,A -85,B 0,C 180,E1 -11073.748,E2 -11073.748} C_VEL
LIN {X 0,Y 399.874,Z 222.457,A -85,B 0,C 180,E1 -11074.789,E2 -11074.789} C_VEL
LIN {X 0,Y 400.523,Z 211.868,A -85,B 0,C 180,E1 -11075.665,E2 -11075.665} C_VEL
LIN {X 0,Y 401.019,Z 200.297,A -85,B 0,C 180,E1 -11076.415,E2 -11076.415} C_VEL
LIN {X 0,Y 401.433,Z 187.174,A -85,B 0,C 180,E1 -11077.039,E2 -11077.039} C_VEL
LIN {X 0,Y 401.755,Z 175.14,A -85,B 0,C 180,E1 -11077.413,E2 -11077.413} C_VEL
LIN {X 0,Y 402.821,Z 88.683,A -85,B 0,C 180,E1 -11078.964,E2 -11078.964} C_VEL
LIN {X 0,Y 400.118,Z 75.203,A -85,B 0,C 180,E1 -11079.327,E2 -11079.327} C_VEL
LIN {X 0,Y 398.381,Z 69.33,A -85,B 0,C 180,E1 -11079.533,E2 -11079.533} C_VEL
LIN {X 0,Y 397.202,Z 63.006,A -85,B 0,C 180,E1 -11081.159,E2 -11081.159} C_VEL
LIN {X 0,Y 397.178,Z 63.011,A -85,B 0,C 180,E1 -11084.343,E2 -11084.343} C_VEL
LIN {X 0,Y 397.176,Z 63.007,A -85,B 0,C 180,E1 -11087.507,E2 -11087.507} C_VEL
LIN {X 0,Y 397.115,Z 63.018,A -85,B 0,C 180,E1 -11090.73,E2 -11090.73} C_VEL
LIN {X 0,Y 397.13,Z 63.017,A -85,B 0,C 180,E1 -11094.019,E2 -11094.019} C_VEL
LIN {X 0,Y 397.196,Z 63.005,A -85,B 0,C 180,E1 -11097.39,E2 -11097.39} C_VEL
LIN {X 0,Y 397.08,Z 63.019,A -85,B 0,C 180,E1 -11100.883,E2 -11100.883} C_VEL
LIN {X 0,Y 397.128,Z 63.014,A -85,B 0,C 180,E1 -11104.493,E2 -11104.493} C_VEL
LIN {X 0,Y 397.109,Z 63.017,A -85,B 0,C 180,E1 -11108.275,E2 -11108.275} C_VEL
LIN {X 0,Y 397.092,Z 63.018,A -85,B 0,C 180,E1 -11110.909,E2 -11110.909} C_VEL
LIN {X 0,Y 397.103,Z 63.022,A -85,B 0,C 180,E1 -11113.649,E2 -11113.649} C_VEL
LIN {X 0,Y 397.104,Z 63.016,A -85,B 0,C 180,E1 -11116.521,E2 -11116.521} C_VEL
LIN {X 0,Y 397.116,Z 63.015,A -85,B 0,C 180,E1 -11120.423,E2 -11120.423} C_VEL
LIN {X 0,Y 397.111,Z 63.016,A -85,B 0,C 180,E1 -11124.266,E2 -11124.266} C_VEL
LIN {X 0,Y 397.118,Z 63.018,A -85,B 0,C 180,E1 -11126.727,E2 -11126.727} C_VEL
LIN {X 0,Y 397.128,Z 63.014,A -85,B 0,C 180,E1 -11130.296,E2 -11130.296} C_VEL
LIN {X 0,Y 397.198,Z 63.009,A -85,B 0,C 180,E1 -11132.61,E2 -11132.61} C_VEL
LIN {X 0,Y 397.137,Z 63.013,A -85,B 0,C 180,E1 -11135.982,E2 -11135.982} C_VEL
LIN {X 0,Y 397.143,Z 63.012,A -85,B 0,C 180,E1 -11139.705,E2 -11139.705} C_VEL
LIN {X 0,Y 397.186,Z 63.009,A -85,B 0,C 180,E1 -11142.845,E2 -11142.845} C_VEL
LIN {X 0,Y 397.233,Z 63.003,A -85,B 0,C 180,E1 -11146.703,E2 -11146.703} C_VEL
LIN {X 0,Y 397.221,Z 63.004,A -85,B 0,C 180,E1 -11149.809,E2 -11149.809} C_VEL
LIN {X 0,Y 397.346,Z 62.987,A -85,B 0,C 180,E1 -11152.888,E2 -11152.888} C_VEL
LIN {X 0,Y 397.256,Z 62.997,A -85,B 0,C 180,E1 -11154.925,E2 -11154.925} C_VEL
LIN {X 0,Y 397.452,Z 62.979,A -85,B 0,C 180,E1 -11157.973,E2 -11157.973} C_VEL
LIN {X 0,Y 397.584,Z 62.962,A -85,B 0,C 180,E1 -11160,E2 -11160} C_VEL
LIN {X 0,Y 397.378,Z 62.983,A -85,B 0,C 180,E1 -11163.042,E2 -11163.042} C_VEL
LIN {X 0,Y 397.338,Z 62.989,A -85,B 0,C 180,E1 -11166.092,E2 -11166.092} C_VEL
LIN {X 0,Y 397.24,Z 63.002,A -85,B 0,C 180,E1 -11169.162,E2 -11169.162} C_VEL
LIN {X 0,Y 397.224,Z 63.002,A -85,B 0,C 180,E1 -11172.258,E2 -11172.258} C_VEL
LIN {X 0,Y 397.184,Z 63.012,A -85,B 0,C 180,E1 -11175.392,E2 -11175.392} C_VEL
LIN {X 0,Y 397.163,Z 63.01,A -85,B 0,C 180,E1 -11178.574,E2 -11178.574} C_VEL
LIN {X 0,Y 397.1,Z 63.017,A -85,B 0,C 180,E1 -11181.818,E2 -11181.818} C_VEL
LIN {X 0,Y 397.127,Z 63.018,A -85,B 0,C 180,E1 -11185.134,E2 -11185.134} C_VEL
LIN {X 0,Y 397.103,Z 63.02,A -85,B 0,C 180,E1 -11188.545,E2 -11188.545} C_VEL
LIN {X 0,Y 397.082,Z 63.02,A -85,B 0,C 180,E1 -11192.071,E2 -11192.071} C_VEL
LIN {X 0,Y 397.122,Z 63.014,A -85,B 0,C 180,E1 -11195.503,E2 -11195.503} C_VEL
LIN {X 0,Y 397.13,Z 63.016,A -85,B 0,C 180,E1 -11198.861,E2 -11198.861} C_VEL
LIN {X 0,Y 397.073,Z 63.026,A -85,B 0,C 180,E1 -11202.267,E2 -11202.267} C_VEL
LIN {X 0,Y 397.09,Z 63.018,A -85,B 0,C 180,E1 -11205.069,E2 -11205.069} C_VEL
LIN {X 0,Y 397.065,Z 63.027,A -85,B 0,C 180,E1 -11208.022,E2 -11208.022} C_VEL
LIN {X 0,Y 397.105,Z 63.016,A -85,B 0,C 180,E1 -11211.143,E2 -11211.143} C_VEL
LIN {X 0,Y 397.121,Z 63.015,A -85,B 0,C 180,E1 -11214.497,E2 -11214.497} C_VEL
LIN {X 0,Y 397.082,Z 63.024,A -85,B 0,C 180,E1 -11217.928,E2 -11217.928} C_VEL
LIN {X 0,Y 397.217,Z 63.157,A -85,B 0,C 180,E1 -11221.355,E2 -11221.355} C_VEL
LIN {X 0,Y 399.648,Z 75.271,A -85,B 0,C 180,E1 -11223.919,E2 -11223.919} C_VEL
LIN {X 0,Y 400.157,Z 79.558,A -85,B 0,C 180,E1 -11224.792,E2 -11224.792} C_VEL
LIN {X 0,Y 398.83,Z 98.99,A -85,B 0,C 180,E1 -11228.533,E2 -11228.533} C_VEL
LIN {X 0,Y 398.279,Z 109.226,A -85,B 0,C 180,E1 -11230.482,E2 -11230.482} C_VEL
LIN {X 0,Y 402.244,Z 141.693,A -85,B 0,C 180,E1 -11231.24,E2 -11231.24} C_VEL
LIN {X 0,Y 401.421,Z 217.968,A -85,B 0,C 180,E1 -11232.619,E2 -11232.619} C_VEL
LIN {X 0,Y 400.873,Z 231.312,A -85,B 0,C 180,E1 -11233.054,E2 -11233.054} C_VEL
LIN {X 0,Y 400.226,Z 244.121,A -85,B 0,C 180,E1 -11233.682,E2 -11233.682} C_VEL
LIN {X 0,Y 399.451,Z 255.478,A -85,B 0,C 180,E1 -11234.436,E2 -11234.436} C_VEL
LIN {X 0,Y 398.68,Z 267.226,A -85,B 0,C 180,E1 -11235.451,E2 -11235.451} C_VEL
LIN {X 0,Y 398.016,Z 277.179,A -85,B 0,C 180,E1 -11236.525,E2 -11236.525} C_VEL
LIN {X 0,Y 397.308,Z 286.418,A -85,B 0,C 180,E1 -11237.744,E2 -11237.744} C_VEL
LIN {X 0,Y 396.754,Z 294.369,A -85,B 0,C 180,E1 -11239.022,E2 -11239.022} C_VEL
LIN {X 0,Y 396.288,Z 302.123,A -85,B 0,C 180,E1 -11240.558,E2 -11240.558} C_VEL
LIN {X 0,Y 396.005,Z 309.271,A -85,B 0,C 180,E1 -11242.351,E2 -11242.351} C_VEL
LIN {X 0,Y 395.793,Z 314.117,A -85,B 0,C 180,E1 -11243.924,E2 -11243.924} C_VEL
LIN {X 0,Y 395.874,Z 317.62,A -85,B 0,C 180,E1 -11245.418,E2 -11245.418} C_VEL
LIN {X 0,Y 395.883,Z 320.199,A -85,B 0,C 180,E1 -11246.947,E2 -11246.947} C_VEL
LIN {X 0,Y 395.923,Z 321.408,A -85,B 0,C 180,E1 -11247.965,E2 -11247.965} C_VEL
LIN {X 0,Y 395.883,Z 322.164,A -85,B 0,C 180,E1 -11248.983,E2 -11248.983} C_VEL
LIN {X 0,Y 395.878,Z 322.521,A -85,B 0,C 180,E1 -11250,E2 -11250} C_VEL
LIN {X 0,Y 395.902,Z 322.069,A -85,B 0,C 180,E1 -11252.035,E2 -11252.035} C_VEL
LIN {X 0,Y 395.823,Z 321.215,A -85,B 0,C 180,E1 -11253.053,E2 -11253.053} C_VEL
LIN {X 0,Y 395.798,Z 319.95,A -85,B 0,C 180,E1 -11254.073,E2 -11254.073} C_VEL
LIN {X 0,Y 395.779,Z 317.002,A -85,B 0,C 180,E1 -11255.736,E2 -11255.736} C_VEL
LIN {X 0,Y 396.03,Z 312.166,A -85,B 0,C 180,E1 -11257.649,E2 -11257.649} C_VEL
LIN {X 0,Y 396.386,Z 305.997,A -85,B 0,C 180,E1 -11259.439,E2 -11259.439} C_VEL
LIN {X 0,Y 396.899,Z 299.292,A -85,B 0,C 180,E1 -11260.973,E2 -11260.973} C_VEL
LIN {X 0,Y 397.804,Z 291.003,A -85,B 0,C 180,E1 -11262.499,E2 -11262.499} C_VEL
LIN {X 0,Y 398.575,Z 281.919,A -85,B 0,C 180,E1 -11263.854,E2 -11263.854} C_VEL
LIN {X 0,Y 399.631,Z 271.045,A -85,B 0,C 180,E1 -11265.152,E2 -11265.152} C_VEL
LIN {X 0,Y 400.696,Z 260.388,A -85,B 0,C 180,E1 -11266.167,E2 -11266.167} C_VEL
LIN {X 0,Y 401.669,Z 248.715,A -85,B 0,C 180,E1 -11267.042,E2 -11267.042} C_VEL
LIN {X 0,Y 402.619,Z 236.609,A -85,B 0,C 180,E1 -11267.721,E2 -11267.721} C_VEL
LIN {X 0,Y 403.407,Z 223.444,A -85,B 0,C 180,E1 -11268.243,E2 -11268.243} C_VEL
LIN {X 0,Y 403.809,Z 209.381,A -85,B 0,C 180,E1 -11268.577,E2 -11268.577} C_VEL
LIN {X 0,Y 404.725,Z 140.66,A -85,B 0,C 180,E1 -11269.819,E2 -11269.819} C_VEL
LIN {X 0,Y 401.009,Z 117.506,A -85,B 0,C 180,E1 -11270.48,E2 -11270.48} C_VEL
LIN {X 0,Y 399.349,Z 108.459,A -85,B 0,C 180,E1 -11270.787,E2 -11270.787} C_VEL
LIN {X 0,Y 400.738,Z 91.078,A -85,B 0,C 180,E1 -11274.222,E2 -11274.222} C_VEL
LIN {X 0,Y 401.377,Z 82.439,A -85,B 0,C 180,E1 -11275.96,E2 -11275.96} C_VEL
LIN {X 0,Y 399.177,Z 71.641,A -85,B 0,C 180,E1 -11278.383,E2 -11278.383} C_VEL
LIN {X 0,Y 397.109,Z 63.017,A -85,B 0,C 180,E1 -11280.448,E2 -11280.448} C_VEL
LIN {X 0,Y 397.121,Z 63.019,A -85,B 0,C 180,E1 -11283.718,E2 -11283.718} C_VEL
LIN {X 0,Y 397.096,Z 63.02,A -85,B 0,C 180,E1 -11287.209,E2 -11287.209} C_VEL
LIN {X 0,Y 397.104,Z 63.018,A -85,B 0,C 180,E1 -11290.445,E2 -11290.445} C_VEL
LIN {X 0,Y 397.104,Z 63.021,A -85,B 0,C 180,E1 -11293.648,E2 -11293.648} C_VEL
LIN {X 0,Y 397.105,Z 63.014,A -85,B 0,C 180,E1 -11296.521,E2 -11296.521} C_VEL
LIN {X 0,Y 397.115,Z 63.01,A -85,B 0,C 180,E1 -11300.423,E2 -11300.423} C_VEL
LIN {X 0,Y 397.11,Z 63.015,A -85,B 0,C 180,E1 -11304.265,E2 -11304.265} C_VEL
LIN {X 0,Y 397.117,Z 63.013,A -85,B 0,C 180,E1 -11306.727,E2 -11306.727} C_VEL
LIN {X 0,Y 397.128,Z 63.01,A -85,B 0,C 180,E1 -11310.296,E2 -11310.296} C_VEL
LIN {X 0,Y 397.198,Z 63.009,A -85,B 0,C 180,E1 -11312.61,E2 -11312.61} C_VEL
LIN {X 0,Y 397.136,Z 63.014,A -85,B 0,C 180,E1 -11315.982,E2 -11315.982} C_VEL
LIN {X 0,Y 397.142,Z 63.011,A -85,B 0,C 180,E1 -11319.705,E2 -11319.705} C_VEL
LIN {X 0,Y 397.185,Z 63.003,A -85,B 0,C 180,E1 -11322.845,E2 -11322.845} C_VEL
LIN {X 0,Y 397.23,Z 63,A -85,B 0,C 180,E1 -11326.679,E2 -11326.679} C_VEL
LIN {X 0,Y 397.221,Z 63.003,A -85,B 0,C 180,E1 -11329.809,E2 -11329.809} C_VEL
LIN {X 0,Y 397.354,Z 62.977,A -85,B 0,C 180,E1 -11332.888,E2 -11332.888} C_VEL
LIN {X 0,Y 397.256,Z 62.998,A -85,B 0,C 180,E1 -11334.925,E2 -11334.925} C_VEL
LIN {X 0,Y 397.451,Z 62.97,A -85,B 0,C 180,E1 -11337.973,E2 -11337.973} C_VEL
LIN {X 0,Y 397.583,Z 62.961,A -85,B 0,C 180,E1 -11340,E2 -11340} C_VEL
LIN {X 0,Y 397.377,Z 62.981,A -85,B 0,C 180,E1 -11343.041,E2 -11343.041} C_VEL
LIN {X 0,Y 397.334,Z 62.989,A -85,B 0,C 180,E1 -11346.613,E2 -11346.613} C_VEL
LIN {X 0,Y 397.239,Z 62.996,A -85,B 0,C 180,E1 -11349.162,E2 -11349.162} C_VEL
LIN {X 0,Y 397.223,Z 63.002,A -85,B 0,C 180,E1 -11352.258,E2 -11352.258} C_VEL
LIN {X 0,Y 397.183,Z 63.011,A -85,B 0,C 180,E1 -11355.392,E2 -11355.392} C_VEL
LIN {X 0,Y 397.161,Z 63.008,A -85,B 0,C 180,E1 -11358.573,E2 -11358.573} C_VEL
LIN {X 0,Y 397.1,Z 63.017,A -85,B 0,C 180,E1 -11361.818,E2 -11361.818} C_VEL
LIN {X 0,Y 397.132,Z 63.017,A -85,B 0,C 180,E1 -11365.133,E2 -11365.133} C_VEL
LIN {X 0,Y 397.102,Z 63.021,A -85,B 0,C 180,E1 -11368.545,E2 -11368.545} C_VEL
LIN {X 0,Y 397.08,Z 63.022,A -85,B 0,C 180,E1 -11372.071,E2 -11372.071} C_VEL
LIN {X 0,Y 397.12,Z 63.016,A -85,B 0,C 180,E1 -11375.503,E2 -11375.503} C_VEL
LIN {X 0,Y 397.101,Z 63.019,A -85,B 0,C 180,E1 -11378.856,E2 -11378.856} C_VEL
LIN {X 0,Y 397.065,Z 63.023,A -85,B 0,C 180,E1 -11382.268,E2 -11382.268} C_VEL
LIN {X 0,Y 397.088,Z 63.022,A -85,B 0,C 180,E1 -11385.069,E2 -11385.069} C_VEL
LIN {X 0,Y 397.062,Z 63.027,A -85,B 0,C 180,E1 -11388.022,E2 -11388.022} C_VEL
LIN {X 0,Y 397.095,Z 63.021,A -85,B 0,C 180,E1 -11391.145,E2 -11391.145} C_VEL
LIN {X 0,Y 397.119,Z 63.02,A -85,B 0,C 180,E1 -11394.497,E2 -11394.497} C_VEL
LIN {X 0,Y 397.17,Z 63.134,A -85,B 0,C 180,E1 -11397.336,E2 -11397.336} C_VEL
LIN {X 0,Y 398.611,Z 70.056,A -85,B 0,C 180,E1 -11399.244,E2 -11399.244} C_VEL
LIN {X 0,Y 403.993,Z 83.953,A -85,B 0,C 180,E1 -11399.852,E2 -11399.852} C_VEL
LIN {X 0,Y 405.507,Z 90.111,A -85,B 0,C 180,E1 -11400.062,E2 -11400.062} C_VEL
LIN {X 0,Y 404.054,Z 176.586,A -85,B 0,C 180,E1 -11401.636,E2 -11401.636} C_VEL
LIN {X 0,Y 403.692,Z 189.96,A -85,B 0,C 180,E1 -11402.092,E2 -11402.092} C_VEL
LIN {X 0,Y 403.158,Z 202.989,A -85,B 0,C 180,E1 -11402.754,E2 -11402.754} C_VEL
LIN {X 0,Y 402.36,Z 214.562,A -85,B 0,C 180,E1 -11403.551,E2 -11403.551} C_VEL
LIN {X 0,Y 401.356,Z 226.32,A -85,B 0,C 180,E1 -11404.595,E2 -11404.595} C_VEL
LIN {X 0,Y 400.413,Z 236.732,A -85,B 0,C 180,E1 -11405.764,E2 -11405.764} C_VEL
LIN {X 0,Y 399.577,Z 245.352,A -85,B 0,C 180,E1 -11406.962,E2 -11406.962} C_VEL
LIN {X 0,Y 398.72,Z 253.148,A -85,B 0,C 180,E1 -11408.275,E2 -11408.275} C_VEL
LIN {X 0,Y 397.888,Z 260.73,A -85,B 0,C 180,E1 -11409.853,E2 -11409.853} C_VEL
LIN {X 0,Y 397.27,Z 266.764,A -85,B 0,C 180,E1 -11411.432,E2 -11411.432} C_VEL
LIN {X 0,Y 396.771,Z 271.57,A -85,B 0,C 180,E1 -11413.039,E2 -11413.039} C_VEL
LIN {X 0,Y 396.382,Z 275.041,A -85,B 0,C 180,E1 -11414.576,E2 -11414.576} C_VEL
LIN {X 0,Y 396.193,Z 276.823,A -85,B 0,C 180,E1 -11415.62,E2 -11415.62} C_VEL
LIN {X 0,Y 396.009,Z 278.885,A -85,B 0,C 180,E1 -11417.445,E2 -11417.445} C_VEL
LIN {X 0,Y 395.892,Z 279.611,A -85,B 0,C 180,E1 -11418.739,E2 -11418.739} C_VEL
LIN {X 0,Y 395.813,Z 279.395,A -85,B 0,C 180,E1 -11420.805,E2 -11420.805} C_VEL
LIN {X 0,Y 395.875,Z 278.702,A -85,B 0,C 180,E1 -11421.835,E2 -11421.835} C_VEL
LIN {X 0,Y 396.075,Z 276.631,A -85,B 0,C 180,E1 -11423.55,E2 -11423.55} C_VEL
LIN {X 0,Y 396.172,Z 272.991,A -85,B 0,C 180,E1 -11425.421,E2 -11425.421} C_VEL
LIN {X 0,Y 396.491,Z 268.855,A -85,B 0,C 180,E1 -11426.952,E2 -11426.952} C_VEL
LIN {X 0,Y 396.797,Z 262.576,A -85,B 0,C 180,E1 -11428.731,E2 -11428.731} C_VEL
LIN {X 0,Y 397.388,Z 255.723,A -85,B 0,C 180,E1 -11430.253,E2 -11430.253} C_VEL
LIN {X 0,Y 397.957,Z 247.171,A -85,B 0,C 180,E1 -11431.771,E2 -11431.771} C_VEL
LIN {X 0,Y 398.553,Z 238.416,A -85,B 0,C 180,E1 -11433.033,E2 -11433.033} C_VEL
LIN {X 0,Y 399.14,Z 232.544,A -85,B 0,C 180,E1 -11433.748,E2 -11433.748} C_VEL
LIN {X 0,Y 398.818,Z 227.962,A -85,B 0,C 180,E1 -11434.283,E2 -11434.283} C_VEL
LIN {X 0,Y 396.557,Z 220.264,A -85,B 0,C 180,E1 -11435.124,E2 -11435.124} C_VEL
LIN {X 0,Y 394.242,Z 212.144,A -85,B 0,C 180,E1 -11435.879,E2 -11435.879} C_VEL
LIN {X 0,Y 393.83,Z 206.899,A -85,B 0,C 180,E1 -11436.272,E2 -11436.272} C_VEL
LIN {X 0,Y 394.359,Z 194.663,A -85,B 0,C 180,E1 -11436.973,E2 -11436.973} C_VEL
LIN {X 0,Y 394.756,Z 182.179,A -85,B 0,C 180,E1 -11437.481,E2 -11437.481} C_VEL
LIN {X 0,Y 394.974,Z 169.364,A -85,B 0,C 180,E1 -11437.798,E2 -11437.798} C_VEL
LIN {X 0,Y 395.985,Z 89.252,A -85,B 0,C 180,E1 -11439.245,E2 -11439.245} C_VEL
LIN {X 0,Y 393.408,Z 76.75,A -85,B 0,C 180,E1 -11439.592,E2 -11439.592} C_VEL
LIN {X 0,Y 391.242,Z 69.763,A -85,B 0,C 180,E1 -11439.826,E2 -11439.826} C_VEL
LIN {X 0,Y 390.161,Z 63.882,A -85,B 0,C 180,E1 -11441.363,E2 -11441.363} C_VEL
LIN {X 0,Y 390.146,Z 63.89,A -85,B 0,C 180,E1 -11444.608,E2 -11444.608} C_VEL
LIN {X 0,Y 390.129,Z 63.886,A -85,B 0,C 180,E1 -11447.833,E2 -11447.833} C_VEL
LIN {X 0,Y 390.063,Z 63.894,A -85,B 0,C 180,E1 -11451.122,E2 -11451.122} C_VEL
LIN {X 0,Y 390.079,Z 63.895,A -85,B 0,C 180,E1 -11454.481,E2 -11454.481} C_VEL
LIN {X 0,Y 390.119,Z 63.891,A -85,B 0,C 180,E1 -11457.93,E2 -11457.93} C_VEL
LIN {X 0,Y 390.026,Z 63.9,A -85,B 0,C 180,E1 -11461.505,E2 -11461.505} C_VEL
LIN {X 0,Y 390.07,Z 63.897,A -85,B 0,C 180,E1 -11464.025,E2 -11464.025} C_VEL
LIN {X 0,Y 390.048,Z 63.9,A -85,B 0,C 180,E1 -11467.552,E2 -11467.552} C_VEL
LIN {X 0,Y 390.059,Z 63.894,A -85,B 0,C 180,E1 -11470.822,E2 -11470.822} C_VEL
LIN {X 0,Y 390.057,Z 63.897,A -85,B 0,C 180,E1 -11473.886,E2 -11473.886} C_VEL
LIN {X 0,Y 390.059,Z 63.895,A -85,B 0,C 180,E1 -11476.79,E2 -11476.79} C_VEL
LIN {X 0,Y 390.059,Z 63.898,A -85,B 0,C 180,E1 -11479.561,E2 -11479.561} C_VEL
LIN {X 0,Y 390.045,Z 63.896,A -85,B 0,C 180,E1 -11482.45,E2 -11482.45} C_VEL
LIN {X 0,Y 390.071,Z 63.893,A -85,B 0,C 180,E1 -11485.976,E2 -11485.976} C_VEL
LIN {X 0,Y 390.05,Z 63.895,A -85,B 0,C 180,E1 -11489.869,E2 -11489.869} C_VEL
LIN {X 0,Y 390.117,Z 63.889,A -85,B 0,C 180,E1 -11493.232,E2 -11493.232} C_VEL
LIN {X 0,Y 390.11,Z 63.894,A -85,B 0,C 180,E1 -11496.751,E2 -11496.751} C_VEL
LIN {X 0,Y 390.108,Z 63.889,A -85,B 0,C 180,E1 -11499.983,E2 -11499.983} C_VEL
LIN {X 0,Y 390.142,Z 63.884,A -85,B 0,C 180,E1 -11503.249,E2 -11503.249} C_VEL
LIN {X 0,Y 390.199,Z 63.881,A -85,B 0,C 180,E1 -11506.562,E2 -11506.562} C_VEL
LIN {X 0,Y 390.172,Z 63.881,A -85,B 0,C 180,E1 -11509.623,E2 -11509.623} C_VEL
LIN {X 0,Y 390.299,Z 63.865,A -85,B 0,C 180,E1 -11512.759,E2 -11512.759} C_VEL
LIN {X 0,Y 390.228,Z 63.873,A -85,B 0,C 180,E1 -11514.834,E2 -11514.834} C_VEL
LIN {X 0,Y 390.421,Z 63.856,A -85,B 0,C 180,E1 -11517.937,E2 -11517.937} C_VEL
LIN {X 0,Y 390.553,Z 63.837,A -85,B 0,C 180,E1 -11520,E2 -11520} C_VEL
LIN {X 0,Y 390.313,Z 63.863,A -85,B 0,C 180,E1 -11523.097,E2 -11523.097} C_VEL
LIN {X 0,Y 390.292,Z 63.866,A -85,B 0,C 180,E1 -11526.203,E2 -11526.203} C_VEL
LIN {X 0,Y 390.198,Z 63.881,A -85,B 0,C 180,E1 -11529.329,E2 -11529.329} C_VEL
LIN {X 0,Y 390.176,Z 63.879,A -85,B 0,C 180,E1 -11532.483,E2 -11532.483} C_VEL
LIN {X 0,Y 390.144,Z 63.886,A -85,B 0,C 180,E1 -11535.677,E2 -11535.677} C_VEL
LIN {X 0,Y 390.107,Z 63.892,A -85,B 0,C 180,E1 -11538.922,E2 -11538.922} C_VEL
LIN {X 0,Y 390.042,Z 63.896,A -85,B 0,C 180,E1 -11542.234,E2 -11542.234} C_VEL
LIN {X 0,Y 390.088,Z 63.891,A -85,B 0,C 180,E1 -11545.733,E2 -11545.733} C_VEL
LIN {X 0,Y 390.048,Z 63.899,A -85,B 0,C 180,E1 -11549.111,E2 -11549.111} C_VEL
LIN {X 0,Y 390.046,Z 63.902,A -85,B 0,C 180,E1 -11552.721,E2 -11552.721} C_VEL
LIN {X 0,Y 390.059,Z 63.894,A -85,B 0,C 180,E1 -11555.825,E2 -11555.825} C_VEL
LIN {X 0,Y 390.071,Z 63.893,A -85,B 0,C 180,E1 -11559.218,E2 -11559.218} C_VEL
LIN {X 0,Y 390.046,Z 63.902,A -85,B 0,C 180,E1 -11562.374,E2 -11562.374} C_VEL
LIN {X 0,Y 390.047,Z 63.896,A -85,B 0,C 180,E1 -11565.354,E2 -11565.354} C_VEL
LIN {X 0,Y 390.027,Z 63.904,A -85,B 0,C 180,E1 -11568.186,E2 -11568.186} C_VEL
LIN {X 0,Y 390.068,Z 63.893,A -85,B 0,C 180,E1 -11570.905,E2 -11570.905} C_VEL
LIN {X 0,Y 390.087,Z 63.89,A -85,B 0,C 180,E1 -11574.793,E2 -11574.793} C_VEL
LIN {X 0,Y 390.026,Z 63.898,A -85,B 0,C 180,E1 -11578.496,E2 -11578.496} C_VEL
LIN {X 0,Y 390.172,Z 64.025,A -85,B 0,C 180,E1 -11581.117,E2 -11581.117} C_VEL
LIN {X 0,Y 392.858,Z 77.48,A -85,B 0,C 180,E1 -11584.017,E2 -11584.017} C_VEL
LIN {X 0,Y 393.149,Z 81.68,A -85,B 0,C 180,E1 -11584.877,E2 -11584.877} C_VEL
LIN {X 0,Y 391.814,Z 100.076,A -85,B 0,C 180,E1 -11588.48,E2 -11588.48} C_VEL
LIN {X 0,Y 391.279,Z 108.778,A -85,B 0,C 180,E1 -11590.174,E2 -11590.174} C_VEL
LIN {X 0,Y 395.414,Z 141.017,A -85,B 0,C 180,E1 -11590.952,E2 -11590.952} C_VEL
LIN {X 0,Y 394.552,Z 218.023,A -85,B 0,C 180,E1 -11592.373,E2 -11592.373} C_VEL
LIN {X 0,Y 393.948,Z 231.991,A -85,B 0,C 180,E1 -11592.847,E2 -11592.847} C_VEL
LIN {X 0,Y 393.252,Z 245.015,A -85,B 0,C 180,E1 -11593.518,E2 -11593.518} C_VEL
LIN {X 0,Y 392.353,Z 257.651,A -85,B 0,C 180,E1 -11594.414,E2 -11594.414} C_VEL
LIN {X 0,Y 391.535,Z 268.928,A -85,B 0,C 180,E1 -11595.445,E2 -11595.445} C_VEL
LIN {X 0,Y 390.934,Z 278.06,A -85,B 0,C 180,E1 -11596.484,E2 -11596.484} C_VEL
LIN {X 0,Y 390.222,Z 287.405,A -85,B 0,C 180,E1 -11597.782,E2 -11597.782} C_VEL
LIN {X 0,Y 389.542,Z 296.476,A -85,B 0,C 180,E1 -11599.343,E2 -11599.343} C_VEL
LIN {X 0,Y 389.113,Z 303.78,A -85,B 0,C 180,E1 -11600.907,E2 -11600.907} C_VEL
LIN {X 0,Y 388.921,Z 308.706,A -85,B 0,C 180,E1 -11602.211,E2 -11602.211} C_VEL
LIN {X 0,Y 388.711,Z 313.952,A -85,B 0,C 180,E1 -11603.943,E2 -11603.943} C_VEL
LIN {X 0,Y 388.8,Z 317.133,A -85,B 0,C 180,E1 -11605.334,E2 -11605.334} C_VEL
LIN {X 0,Y 388.785,Z 319.744,A -85,B 0,C 180,E1 -11606.891,E2 -11606.891} C_VEL
LIN {X 0,Y 388.853,Z 320.973,A -85,B 0,C 180,E1 -11607.928,E2 -11607.928} C_VEL
LIN {X 0,Y 388.81,Z 321.758,A -85,B 0,C 180,E1 -11608.964,E2 -11608.964} C_VEL
LIN {X 0,Y 388.802,Z 322.129,A -85,B 0,C 180,E1 -11610,E2 -11610} C_VEL
LIN {X 0,Y 388.814,Z 321.707,A -85,B 0,C 180,E1 -11612.072,E2 -11612.072} C_VEL
LIN {X 0,Y 388.723,Z 320.883,A -85,B 0,C 180,E1 -11613.109,E2 -11613.109} C_VEL
LIN {X 0,Y 388.718,Z 319.634,A -85,B 0,C 180,E1 -11614.147,E2 -11614.147} C_VEL
LIN {X 0,Y 388.727,Z 316.225,A -85,B 0,C 180,E1 -11616.078,E2 -11616.078} C_VEL
LIN {X 0,Y 388.963,Z 311.919,A -85,B 0,C 180,E1 -11617.788,E2 -11617.788} C_VEL
LIN {X 0,Y 389.342,Z 305.807,A -85,B 0,C 180,E1 -11619.612,E2 -11619.612} C_VEL
LIN {X 0,Y 389.91,Z 299.149,A -85,B 0,C 180,E1 -11621.173,E2 -11621.173} C_VEL
LIN {X 0,Y 390.848,Z 290.914,A -85,B 0,C 180,E1 -11622.725,E2 -11622.725} C_VEL
LIN {X 0,Y 391.626,Z 282.386,A -85,B 0,C 180,E1 -11624.039,E2 -11624.039} C_VEL
LIN {X 0,Y 392.68,Z 272.19,A -85,B 0,C 180,E1 -11625.307,E2 -11625.307} C_VEL
LIN {X 0,Y 393.902,Z 260.58,A -85,B 0,C 180,E1 -11626.454,E2 -11626.454} C_VEL
LIN {X 0,Y 394.912,Z 249.127,A -85,B 0,C 180,E1 -11627.343,E2 -11627.343} C_VEL
LIN {X 0,Y 395.998,Z 235.994,A -85,B 0,C 180,E1 -11628.094,E2 -11628.094} C_VEL
LIN {X 0,Y 396.805,Z 222.745,A -85,B 0,C 180,E1 -11628.624,E2 -11628.624} C_VEL
LIN {X 0,Y 397.182,Z 209.757,A -85,B 0,C 180,E1 -11628.94,E2 -11628.94} C_VEL
LIN {X 0,Y 398.137,Z 141.437,A -85,B 0,C 180,E1 -11630.195,E2 -11630.195} C_VEL
LIN {X 0,Y 394.798,Z 120.291,A -85,B 0,C 180,E1 -11630.812,E2 -11630.812} C_VEL
LIN {X 0,Y 392.539,Z 108.079,A -85,B 0,C 180,E1 -11631.222,E2 -11631.222} C_VEL
LIN {X 0,Y 394.082,Z 90.182,A -85,B 0,C 180,E1 -11634.829,E2 -11634.829} C_VEL
LIN {X 0,Y 394.565,Z 85.064,A -85,B 0,C 180,E1 -11635.874,E2 -11635.874} C_VEL
LIN {X 0,Y 393.167,Z 76.971,A -85,B 0,C 180,E1 -11637.695,E2 -11637.695} C_VEL
LIN {X 0,Y 390.058,Z 63.893,A -85,B 0,C 180,E1 -11640.822,E2 -11640.822} C_VEL
LIN {X 0,Y 390.07,Z 63.897,A -85,B 0,C 180,E1 -11644.025,E2 -11644.025} C_VEL
LIN {X 0,Y 390.046,Z 63.9,A -85,B 0,C 180,E1 -11647.551,E2 -11647.551} C_VEL
LIN {X 0,Y 390.059,Z 63.895,A -85,B 0,C 180,E1 -11650.821,E2 -11650.821} C_VEL
LIN {X 0,Y 390.057,Z 63.895,A -85,B 0,C 180,E1 -11653.886,E2 -11653.886} C_VEL
LIN {X 0,Y 390.06,Z 63.892,A -85,B 0,C 180,E1 -11656.79,E2 -11656.79} C_VEL
LIN {X 0,Y 390.059,Z 63.892,A -85,B 0,C 180,E1 -11659.561,E2 -11659.561} C_VEL
LIN {X 0,Y 390.045,Z 63.893,A -85,B 0,C 180,E1 -11662.449,E2 -11662.449} C_VEL
LIN {X 0,Y 390.071,Z 63.889,A -85,B 0,C 180,E1 -11665.975,E2 -11665.975} C_VEL
LIN {X 0,Y 390.05,Z 63.892,A -85,B 0,C 180,E1 -11669.869,E2 -11669.869} C_VEL
LIN {X 0,Y 390.117,Z 63.886,A -85,B 0,C 180,E1 -11673.232,E2 -11673.232} C_VEL
LIN {X 0,Y 390.11,Z 63.892,A -85,B 0,C 180,E1 -11676.75,E2 -11676.75} C_VEL
LIN {X 0,Y 390.107,Z 63.888,A -85,B 0,C 180,E1 -11679.983,E2 -11679.983} C_VEL
LIN {X 0,Y 390.142,Z 63.88,A -85,B 0,C 180,E1 -11683.248,E2 -11683.248} C_VEL
LIN {X 0,Y 390.198,Z 63.877,A -85,B 0,C 180,E1 -11686.561,E2 -11686.561} C_VEL
LIN {X 0,Y 390.209,Z 63.878,A -85,B 0,C 180,E1 -11690.671,E2 -11690.671} C_VEL
LIN {X 0,Y 390.329,Z 63.855,A -85,B 0,C 180,E1 -11693.798,E2 -11693.798} C_VEL
LIN {X 0,Y 390.42,Z 63.846,A -85,B 0,C 180,E1 -11697.937,E2 -11697.937} C_VEL
LIN {X 0,Y 390.552,Z 63.836,A -85,B 0,C 180,E1 -11700,E2 -11700} C_VEL
LIN {X 0,Y 390.312,Z 63.861,A -85,B 0,C 180,E1 -11703.096,E2 -11703.096} C_VEL
LIN {X 0,Y 390.289,Z 63.867,A -85,B 0,C 180,E1 -11706.606,E2 -11706.606} C_VEL
LIN {X 0,Y 390.196,Z 63.874,A -85,B 0,C 180,E1 -11709.329,E2 -11709.329} C_VEL
LIN {X 0,Y 390.174,Z 63.88,A -85,B 0,C 180,E1 -11712.483,E2 -11712.483} C_VEL
LIN {X 0,Y 390.143,Z 63.887,A -85,B 0,C 180,E1 -11715.677,E2 -11715.677} C_VEL
LIN {X 0,Y 390.105,Z 63.886,A -85,B 0,C 180,E1 -11718.922,E2 -11718.922} C_VEL
LIN {X 0,Y 390.043,Z 63.897,A -85,B 0,C 180,E1 -11722.234,E2 -11722.234} C_VEL
LIN {X 0,Y 390.083,Z 63.892,A -85,B 0,C 180,E1 -11725.62,E2 -11725.62} C_VEL
LIN {X 0,Y 390.046,Z 63.898,A -85,B 0,C 180,E1 -11729.11,E2 -11729.11} C_VEL
LIN {X 0,Y 390.045,Z 63.9,A -85,B 0,C 180,E1 -11732.721,E2 -11732.721} C_VEL
LIN {X 0,Y 390.057,Z 63.898,A -85,B 0,C 180,E1 -11735.825,E2 -11735.825} C_VEL
LIN {X 0,Y 390.043,Z 63.897,A -85,B 0,C 180,E1 -11739.213,E2 -11739.213} C_VEL
LIN {X 0,Y 390.04,Z 63.899,A -85,B 0,C 180,E1 -11742.373,E2 -11742.373} C_VEL
LIN {X 0,Y 390.045,Z 63.901,A -85,B 0,C 180,E1 -11745.354,E2 -11745.354} C_VEL
LIN {X 0,Y 390.028,Z 63.903,A -85,B 0,C 180,E1 -11748.186,E2 -11748.186} C_VEL
LIN {X 0,Y 390.06,Z 63.897,A -85,B 0,C 180,E1 -11750.904,E2 -11750.904} C_VEL
LIN {X 0,Y 390.085,Z 63.897,A -85,B 0,C 180,E1 -11754.793,E2 -11754.793} C_VEL
LIN {X 0,Y 390.114,Z 64.054,A -85,B 0,C 180,E1 -11756.978,E2 -11756.978} C_VEL
LIN {X 0,Y 391.496,Z 70.367,A -85,B 0,C 180,E1 -11758.764,E2 -11758.764} C_VEL
LIN {X 0,Y 397.717,Z 86.124,A -85,B 0,C 180,E1 -11759.499,E2 -11759.499} C_VEL
LIN {X 0,Y 398.955,Z 91.182,A -85,B 0,C 180,E1 -11759.676,E2 -11759.676} C_VEL
LIN {X 0,Y 397.471,Z 177.073,A -85,B 0,C 180,E1 -11761.267,E2 -11761.267} C_VEL
LIN {X 0,Y 397.066,Z 190.677,A -85,B 0,C 180,E1 -11761.74,E2 -11761.74} C_VEL
LIN {X 0,Y 396.518,Z 203.401,A -85,B 0,C 180,E1 -11762.401,E2 -11762.401} C_VEL
LIN {X 0,Y 395.688,Z 214.976,A -85,B 0,C 180,E1 -11763.211,E2 -11763.211} C_VEL
LIN {X 0,Y 394.626,Z 226.725,A -85,B 0,C 180,E1 -11764.272,E2 -11764.272} C_VEL
LIN {X 0,Y 393.604,Z 237.437,A -85,B 0,C 180,E1 -11765.5,E2 -11765.5} C_VEL
LIN {X 0,Y 392.665,Z 246.578,A -85,B 0,C 180,E1 -11766.811,E2 -11766.811} C_VEL
LIN {X 0,Y 391.612,Z 255.611,A -85,B 0,C 180,E1 -11768.414,E2 -11768.414} C_VEL
LIN {X 0,Y 390.788,Z 262.779,A -85,B 0,C 180,E1 -11770.02,E2 -11770.02} C_VEL
LIN {X 0,Y 390.127,Z 268.441,A -85,B 0,C 180,E1 -11771.624,E2 -11771.624} C_VEL
LIN {X 0,Y 389.639,Z 272.847,A -85,B 0,C 180,E1 -11773.226,E2 -11773.226} C_VEL
LIN {X 0,Y 389.383,Z 275.16,A -85,B 0,C 180,E1 -11774.292,E2 -11774.292} C_VEL
LIN {X 0,Y 389.159,Z 277.023,A -85,B 0,C 180,E1 -11775.355,E2 -11775.355} C_VEL
LIN {X 0,Y 388.942,Z 279.279,A -85,B 0,C 180,E1 -11777.358,E2 -11777.358} C_VEL
LIN {X 0,Y 388.812,Z 279.945,A -85,B 0,C 180,E1 -11778.531,E2 -11778.531} C_VEL
LIN {X 0,Y 388.73,Z 280.108,A -85,B 0,C 180,E1 -11779.584,E2 -11779.584} C_VEL
LIN {X 0,Y 388.79,Z 279.188,A -85,B 0,C 180,E1 -11781.685,E2 -11781.685} C_VEL
LIN {X 0,Y 389.008,Z 277.041,A -85,B 0,C 180,E1 -11783.543,E2 -11783.543} C_VEL
LIN {X 0,Y 389.082,Z 273.685,A -85,B 0,C 180,E1 -11785.338,E2 -11785.338} C_VEL
LIN {X 0,Y 389.399,Z 269.64,A -85,B 0,C 180,E1 -11786.896,E2 -11786.896} C_VEL
LIN {X 0,Y 389.722,Z 263.458,A -85,B 0,C 180,E1 -11788.708,E2 -11788.708} C_VEL
LIN {X 0,Y 390.326,Z 256.714,A -85,B 0,C 180,E1 -11790.258,E2 -11790.258} C_VEL
LIN {X 0,Y 390.917,Z 248.353,A -85,B 0,C 180,E1 -11791.803,E2 -11791.803} C_VEL
LIN {X 0,Y 391.514,Z 239.757,A -85,B 0,C 180,E1 -11793.087,E2 -11793.087} C_VEL
LIN {X 0,Y 392.378,Z 230.297,A -85,B 0,C 180,E1 -11794.237,E2 -11794.237} C_VEL
LIN {X 0,Y 393.197,Z 218.596,A -85,B 0,C 180,E1 -11795.385,E2 -11795.385} C_VEL
LIN {X 0,Y 393.83,Z 206.899,A -85,B 0,C 180,E1 -11796.272,E2 -11796.272} C_VEL
LIN {X 0,Y 393.43,Z 201.546,A -85,B 0,C 180,E1 -11796.634,E2 -11796.634} C_VEL
LIN {X 0,Y 391.015,Z 192.744,A -85,B 0,C 180,E1 -11797.203,E2 -11797.203} C_VEL
LIN {X 0,Y 388.543,Z 183.715,A -85,B 0,C 180,E1 -11797.675,E2 -11797.675} C_VEL
LIN {X 0,Y 387.985,Z 178.01,A -85,B 0,C 180,E1 -11797.878,E2 -11797.878} C_VEL
LIN {X 0,Y 388.727,Z 128.523,A -85,B 0,C 180,E1 -11798.819,E2 -11798.819} C_VEL
LIN {X 0,Y 389.106,Z 89.612,A -85,B 0,C 180,E1 -11799.54,E2 -11799.54} C_VEL
LIN {X 0,Y 386.725,Z 78.344,A -85,B 0,C 180,E1 -11799.862,E2 -11799.862} C_VEL
LIN {X 0,Y 384.096,Z 70.084,A -85,B 0,C 180,E1 -11800.16,E2 -11800.16} C_VEL
LIN {X 0,Y 383.121,Z 64.758,A -85,B 0,C 180,E1 -11801.574,E2 -11801.574} C_VEL
LIN {X 0,Y 383.112,Z 64.762,A -85,B 0,C 180,E1 -11804.882,E2 -11804.882} C_VEL
LIN {X 0,Y 383.091,Z 64.766,A -85,B 0,C 180,E1 -11808.172,E2 -11808.172} C_VEL
LIN {X 0,Y 382.997,Z 64.774,A -85,B 0,C 180,E1 -11811.531,E2 -11811.531} C_VEL
LIN {X 0,Y 383.052,Z 64.767,A -85,B 0,C 180,E1 -11814.961,E2 -11814.961} C_VEL
LIN {X 0,Y 383.054,Z 64.771,A -85,B 0,C 180,E1 -11818.277,E2 -11818.277} C_VEL
LIN {X 0,Y 383.012,Z 64.776,A -85,B 0,C 180,E1 -11822.15,E2 -11822.15} C_VEL
LIN {X 0,Y 383.02,Z 64.771,A -85,B 0,C 180,E1 -11824.668,E2 -11824.668} C_VEL
LIN {X 0,Y 383.004,Z 64.777,A -85,B 0,C 180,E1 -11827.905,E2 -11827.905} C_VEL
LIN {X 0,Y 382.987,Z 64.779,A -85,B 0,C 180,E1 -11831.348,E2 -11831.348} C_VEL
LIN {X 0,Y 382.998,Z 64.774,A -85,B 0,C 180,E1 -11834.304,E2 -11834.304} C_VEL
LIN {X 0,Y 383.012,Z 64.777,A -85,B 0,C 180,E1 -11837.24,E2 -11837.24} C_VEL
LIN {X 0,Y 383.017,Z 64.771,A -85,B 0,C 180,E1 -11840.414,E2 -11840.414} C_VEL
LIN {X 0,Y 383.028,Z 64.77,A -85,B 0,C 180,E1 -11844.045,E2 -11844.045} C_VEL
LIN {X 0,Y 382.99,Z 64.776,A -85,B 0,C 180,E1 -11847.578,E2 -11847.578} C_VEL
LIN {X 0,Y 382.996,Z 64.775,A -85,B 0,C 180,E1 -11850.301,E2 -11850.301} C_VEL
LIN {X 0,Y 383.084,Z 64.763,A -85,B 0,C 180,E1 -11854.021,E2 -11854.021} C_VEL
LIN {X 0,Y 383.016,Z 64.772,A -85,B 0,C 180,E1 -11857.336,E2 -11857.336} C_VEL
LIN {X 0,Y 383.064,Z 64.77,A -85,B 0,C 180,E1 -11860.717,E2 -11860.717} C_VEL
LIN {X 0,Y 383.085,Z 64.765,A -85,B 0,C 180,E1 -11864.027,E2 -11864.027} C_VEL
LIN {X 0,Y 383.141,Z 64.756,A -85,B 0,C 180,E1 -11867.284,E2 -11867.284} C_VEL
LIN {X 0,Y 383.151,Z 64.758,A -85,B 0,C 180,E1 -11870.498,E2 -11870.498} C_VEL
LIN {X 0,Y 383.252,Z 64.744,A -85,B 0,C 180,E1 -11872.625,E2 -11872.625} C_VEL
LIN {X 0,Y 383.2,Z 64.749,A -85,B 0,C 180,E1 -11874.739,E2 -11874.739} C_VEL
LIN {X 0,Y 383.388,Z 64.731,A -85,B 0,C 180,E1 -11877.899,E2 -11877.899} C_VEL
LIN {X 0,Y 383.523,Z 64.713,A -85,B 0,C 180,E1 -11880,E2 -11880} C_VEL
LIN {X 0,Y 383.249,Z 64.743,A -85,B 0,C 180,E1 -11883.154,E2 -11883.154} C_VEL
LIN {X 0,Y 383.248,Z 64.743,A -85,B 0,C 180,E1 -11886.317,E2 -11886.317} C_VEL
LIN {X 0,Y 383.148,Z 64.762,A -85,B 0,C 180,E1 -11889.502,E2 -11889.502} C_VEL
LIN {X 0,Y 383.141,Z 64.756,A -85,B 0,C 180,E1 -11892.716,E2 -11892.716} C_VEL
LIN {X 0,Y 383.085,Z 64.763,A -85,B 0,C 180,E1 -11895.973,E2 -11895.973} C_VEL
LIN {X 0,Y 383.063,Z 64.771,A -85,B 0,C 180,E1 -11899.284,E2 -11899.284} C_VEL
LIN {X 0,Y 382.999,Z 64.776,A -85,B 0,C 180,E1 -11902.666,E2 -11902.666} C_VEL
LIN {X 0,Y 383.041,Z 64.769,A -85,B 0,C 180,E1 -11906.126,E2 -11906.126} C_VEL
LIN {X 0,Y 382.988,Z 64.775,A -85,B 0,C 180,E1 -11909.7,E2 -11909.7} C_VEL
LIN {X 0,Y 383.007,Z 64.773,A -85,B 0,C 180,E1 -11913.401,E2 -11913.401} C_VEL
LIN {X 0,Y 383.035,Z 64.771,A -85,B 0,C 180,E1 -11916.164,E2 -11916.164} C_VEL
LIN {X 0,Y 383.011,Z 64.774,A -85,B 0,C 180,E1 -11919.958,E2 -11919.958} C_VEL
LIN {X 0,Y 383.009,Z 64.774,A -85,B 0,C 180,E1 -11922.778,E2 -11922.778} C_VEL
LIN {X 0,Y 383,Z 64.776,A -85,B 0,C 180,E1 -11925.789,E2 -11925.789} C_VEL
LIN {X 0,Y 382.973,Z 64.777,A -85,B 0,C 180,E1 -11928.799,E2 -11928.799} C_VEL
LIN {X 0,Y 382.998,Z 64.779,A -85,B 0,C 180,E1 -11932.097,E2 -11932.097} C_VEL
LIN {X 0,Y 383.021,Z 64.772,A -85,B 0,C 180,E1 -11935.332,E2 -11935.332} C_VEL
LIN {X 0,Y 382.986,Z 64.776,A -85,B 0,C 180,E1 -11939.081,E2 -11939.081} C_VEL
LIN {X 0,Y 383.092,Z 64.91,A -85,B 0,C 180,E1 -11940.874,E2 -11940.874} C_VEL
LIN {X 0,Y 385.721,Z 77.789,A -85,B 0,C 180,E1 -11943.712,E2 -11943.712} C_VEL
LIN {X 0,Y 386.199,Z 82.39,A -85,B 0,C 180,E1 -11944.681,E2 -11944.681} C_VEL
LIN {X 0,Y 384.843,Z 100.51,A -85,B 0,C 180,E1 -11948.296,E2 -11948.296} C_VEL
LIN {X 0,Y 384.326,Z 108.312,A -85,B 0,C 180,E1 -11949.845,E2 -11949.845} C_VEL
LIN {X 0,Y 388.595,Z 142.119,A -85,B 0,C 180,E1 -11950.691,E2 -11950.691} C_VEL
LIN {X 0,Y 387.691,Z 218.035,A -85,B 0,C 180,E1 -11952.119,E2 -11952.119} C_VEL
LIN {X 0,Y 387.055,Z 231.872,A -85,B 0,C 180,E1 -11952.6,E2 -11952.6} C_VEL
LIN {X 0,Y 386.337,Z 244.808,A -85,B 0,C 180,E1 -11953.282,E2 -11953.282} C_VEL
LIN {X 0,Y 385.449,Z 256.607,A -85,B 0,C 180,E1 -11954.127,E2 -11954.127} C_VEL
LIN {X 0,Y 384.64,Z 268.011,A -85,B 0,C 180,E1 -11955.179,E2 -11955.179} C_VEL
LIN {X 0,Y 383.895,Z 278.276,A -85,B 0,C 180,E1 -11956.367,E2 -11956.367} C_VEL
LIN {X 0,Y 383.118,Z 288.334,A -85,B 0,C 180,E1 -11957.821,E2 -11957.821} C_VEL
LIN {X 0,Y 382.392,Z 297.177,A -85,B 0,C 180,E1 -11959.409,E2 -11959.409} C_VEL
LIN {X 0,Y 382.007,Z 304.233,A -85,B 0,C 180,E1 -11961.003,E2 -11961.003} C_VEL
LIN {X 0,Y 381.792,Z 309.879,A -85,B 0,C 180,E1 -11962.596,E2 -11962.596} C_VEL
LIN {X 0,Y 381.634,Z 313.752,A -85,B 0,C 180,E1 -11963.957,E2 -11963.957} C_VEL
LIN {X 0,Y 381.686,Z 317.635,A -85,B 0,C 180,E1 -11965.776,E2 -11965.776} C_VEL
LIN {X 0,Y 381.785,Z 320.534,A -85,B 0,C 180,E1 -11967.89,E2 -11967.89} C_VEL
LIN {X 0,Y 381.74,Z 321.35,A -85,B 0,C 180,E1 -11968.945,E2 -11968.945} C_VEL
LIN {X 0,Y 381.728,Z 321.737,A -85,B 0,C 180,E1 -11970,E2 -11970} C_VEL
LIN {X 0,Y 381.72,Z 321.734,A -85,B 0,C 180,E1 -11971.055,E2 -11971.055} C_VEL
LIN {X 0,Y 381.727,Z 321.345,A -85,B 0,C 180,E1 -11972.11,E2 -11972.11} C_VEL
LIN {X 0,Y 381.627,Z 320.551,A -85,B 0,C 180,E1 -11973.167,E2 -11973.167} C_VEL
LIN {X 0,Y 381.639,Z 319.321,A -85,B 0,C 180,E1 -11974.224,E2 -11974.224} C_VEL
LIN {X 0,Y 381.625,Z 316.277,A -85,B 0,C 180,E1 -11976.029,E2 -11976.029} C_VEL
LIN {X 0,Y 381.887,Z 311.675,A -85,B 0,C 180,E1 -11977.934,E2 -11977.934} C_VEL
LIN {X 0,Y 382.225,Z 306.595,A -85,B 0,C 180,E1 -11979.525,E2 -11979.525} C_VEL
LIN {X 0,Y 382.794,Z 300.242,A -85,B 0,C 180,E1 -11981.115,E2 -11981.115} C_VEL
LIN {X 0,Y 383.748,Z 292.322,A -85,B 0,C 180,E1 -11982.696,E2 -11982.696} C_VEL
LIN {X 0,Y 384.588,Z 283.701,A -85,B 0,C 180,E1 -11984.1,E2 -11984.1} C_VEL
LIN {X 0,Y 385.705,Z 273.43,A -85,B 0,C 180,E1 -11985.455,E2 -11985.455} C_VEL
LIN {X 0,Y 386.945,Z 262.216,A -85,B 0,C 180,E1 -11986.622,E2 -11986.622} C_VEL
LIN {X 0,Y 388.006,Z 251.262,A -85,B 0,C 180,E1 -11987.526,E2 -11987.526} C_VEL
LIN {X 0,Y 389.073,Z 239.157,A -85,B 0,C 180,E1 -11988.292,E2 -11988.292} C_VEL
LIN {X 0,Y 389.996,Z 226.616,A -85,B 0,C 180,E1 -11988.859,E2 -11988.859} C_VEL
LIN {X 0,Y 390.469,Z 213.597,A -85,B 0,C 180,E1 -11989.245,E2 -11989.245} C_VEL
LIN {X 0,Y 391.554,Z 141.717,A -85,B 0,C 180,E1 -11990.596,E2 -11990.596} C_VEL
LIN {X 0,Y 387.971,Z 119.404,A -85,B 0,C 180,E1 -11991.269,E2 -11991.269} C_VEL
LIN {X 0,Y 385.721,Z 107.665,A -85,B 0,C 180,E1 -11991.682,E2 -11991.682} C_VEL
LIN {X 0,Y 387.165,Z 91.833,A -85,B 0,C 180,E1 -11994.935,E2 -11994.935} C_VEL
LIN {X 0,Y 387.688,Z 86.339,A -85,B 0,C 180,E1 -11996.079,E2 -11996.079} C_VEL
LIN {X 0,Y 385.917,Z 76.922,A -85,B 0,C 180,E1 -11998.261,E2 -11998.261} C_VEL
LIN {X 0,Y 382.993,Z 64.774,A -85,B 0,C 180,E1 -12001.263,E2 -12001.263} C_VEL
LIN {X 0,Y 383.02,Z 64.775,A -85,B 0,C 180,E1 -12004.668,E2 -12004.668} C_VEL
LIN {X 0,Y 383.002,Z 64.777,A -85,B 0,C 180,E1 -12007.904,E2 -12007.904} C_VEL
LIN {X 0,Y 382.987,Z 64.778,A -85,B 0,C 180,E1 -12011.347,E2 -12011.347} C_VEL
LIN {X 0,Y 382.998,Z 64.771,A -85,B 0,C 180,E1 -12014.303,E2 -12014.303} C_VEL
LIN {X 0,Y 383.013,Z 64.77,A -85,B 0,C 180,E1 -12017.24,E2 -12017.24} C_VEL
LIN {X 0,Y 383.016,Z 64.766,A -85,B 0,C 180,E1 -12020.414,E2 -12020.414} C_VEL
LIN {X 0,Y 383.027,Z 64.769,A -85,B 0,C 180,E1 -12024.044,E2 -12024.044} C_VEL
LIN {X 0,Y 382.99,Z 64.778,A -85,B 0,C 180,E1 -12027.578,E2 -12027.578} C_VEL
LIN {X 0,Y 382.995,Z 64.771,A -85,B 0,C 180,E1 -12030.3,E2 -12030.3} C_VEL
LIN {X 0,Y 383.06,Z 64.771,A -85,B 0,C 180,E1 -12032.698,E2 -12032.698} C_VEL
LIN {X 0,Y 383.056,Z 64.769,A -85,B 0,C 180,E1 -12035.04,E2 -12035.04} C_VEL
LIN {X 0,Y 382.997,Z 64.771,A -85,B 0,C 180,E1 -12038.469,E2 -12038.469} C_VEL
LIN {X 0,Y 383.066,Z 64.765,A -85,B 0,C 180,E1 -12041.826,E2 -12041.826} C_VEL
LIN {X 0,Y 383.114,Z 64.761,A -85,B 0,C 180,E1 -12045.118,E2 -12045.118} C_VEL
LIN {X 0,Y 383.101,Z 64.758,A -85,B 0,C 180,E1 -12048.358,E2 -12048.358} C_VEL
LIN {X 0,Y 383.267,Z 64.741,A -85,B 0,C 180,E1 -12051.976,E2 -12051.976} C_VEL
LIN {X 0,Y 383.2,Z 64.75,A -85,B 0,C 180,E1 -12054.738,E2 -12054.738} C_VEL
LIN {X 0,Y 383.387,Z 64.722,A -85,B 0,C 180,E1 -12057.899,E2 -12057.899} C_VEL
LIN {X 0,Y 383.521,Z 64.712,A -85,B 0,C 180,E1 -12060,E2 -12060} C_VEL
LIN {X 0,Y 383.248,Z 64.741,A -85,B 0,C 180,E1 -12063.154,E2 -12063.154} C_VEL
LIN {X 0,Y 383.25,Z 64.743,A -85,B 0,C 180,E1 -12066.595,E2 -12066.595} C_VEL
LIN {X 0,Y 383.146,Z 64.753,A -85,B 0,C 180,E1 -12069.502,E2 -12069.502} C_VEL
LIN {X 0,Y 383.14,Z 64.757,A -85,B 0,C 180,E1 -12072.716,E2 -12072.716} C_VEL
LIN {X 0,Y 383.084,Z 64.765,A -85,B 0,C 180,E1 -12075.973,E2 -12075.973} C_VEL
LIN {X 0,Y 383.061,Z 64.766,A -85,B 0,C 180,E1 -12079.284,E2 -12079.284} C_VEL
LIN {X 0,Y 383.011,Z 64.772,A -85,B 0,C 180,E1 -12082.665,E2 -12082.665} C_VEL
LIN {X 0,Y 383.042,Z 64.77,A -85,B 0,C 180,E1 -12086.126,E2 -12086.126} C_VEL
LIN {X 0,Y 382.986,Z 64.776,A -85,B 0,C 180,E1 -12089.7,E2 -12089.7} C_VEL
LIN {X 0,Y 383.005,Z 64.773,A -85,B 0,C 180,E1 -12093.4,E2 -12093.4} C_VEL
LIN {X 0,Y 383.033,Z 64.775,A -85,B 0,C 180,E1 -12096.164,E2 -12096.164} C_VEL
LIN {X 0,Y 382.989,Z 64.772,A -85,B 0,C 180,E1 -12099.961,E2 -12099.961} C_VEL
LIN {X 0,Y 383.006,Z 64.777,A -85,B 0,C 180,E1 -12102.778,E2 -12102.778} C_VEL
LIN {X 0,Y 382.998,Z 64.78,A -85,B 0,C 180,E1 -12105.789,E2 -12105.789} C_VEL
LIN {X 0,Y 382.986,Z 64.779,A -85,B 0,C 180,E1 -12108.796,E2 -12108.796} C_VEL
LIN {X 0,Y 382.994,Z 64.779,A -85,B 0,C 180,E1 -12112.097,E2 -12112.097} C_VEL
LIN {X 0,Y 383.018,Z 64.778,A -85,B 0,C 180,E1 -12115.332,E2 -12115.332} C_VEL
LIN {X 0,Y 383.076,Z 64.838,A -85,B 0,C 180,E1 -12116.567,E2 -12116.567} C_VEL
LIN {X 0,Y 384.378,Z 70.905,A -85,B 0,C 180,E1 -12118.299,E2 -12118.299} C_VEL
LIN {X 0,Y 391.392,Z 88.102,A -85,B 0,C 180,E1 -12119.125,E2 -12119.125} C_VEL
LIN {X 0,Y 392.496,Z 92.912,A -85,B 0,C 180,E1 -12119.293,E2 -12119.293} C_VEL
LIN {X 0,Y 390.892,Z 177.787,A -85,B 0,C 180,E1 -12120.891,E2 -12120.891} C_VEL
LIN {X 0,Y 390.469,Z 191.154,A -85,B 0,C 180,E1 -12121.366,E2 -12121.366} C_VEL
LIN {X 0,Y 389.884,Z 204.07,A -85,B 0,C 180,E1 -12122.052,E2 -12122.052} C_VEL
LIN {X 0,Y 389.02,Z 215.529,A -85,B 0,C 180,E1 -12122.871,E2 -12122.871} C_VEL
LIN {X 0,Y 387.915,Z 227.142,A -85,B 0,C 180,E1 -12123.938,E2 -12123.938} C_VEL
LIN {X 0,Y 386.857,Z 237.639,A -85,B 0,C 180,E1 -12125.158,E2 -12125.158} C_VEL
LIN {X 0,Y 385.925,Z 246.149,A -85,B 0,C 180,E1 -12126.382,E2 -12126.382} C_VEL
LIN {X 0,Y 384.814,Z 255.321,A -85,B 0,C 180,E1 -12128.013,E2 -12128.013} C_VEL
LIN {X 0,Y 383.921,Z 262.649,A -85,B 0,C 180,E1 -12129.646,E2 -12129.646} C_VEL
LIN {X 0,Y 383.218,Z 268.425,A -85,B 0,C 180,E1 -12131.28,E2 -12131.28} C_VEL
LIN {X 0,Y 382.685,Z 272.925,A -85,B 0,C 180,E1 -12132.912,E2 -12132.912} C_VEL
LIN {X 0,Y 382.381,Z 275.282,A -85,B 0,C 180,E1 -12133.997,E2 -12133.997} C_VEL
LIN {X 0,Y 382.153,Z 277.195,A -85,B 0,C 180,E1 -12135.08,E2 -12135.08} C_VEL
LIN {X 0,Y 381.944,Z 278.649,A -85,B 0,C 180,E1 -12136.16,E2 -12136.16} C_VEL
LIN {X 0,Y 381.879,Z 279.673,A -85,B 0,C 180,E1 -12137.265,E2 -12137.265} C_VEL
LIN {X 0,Y 381.666,Z 280.499,A -85,B 0,C 180,E1 -12139.389,E2 -12139.389} C_VEL
LIN {X 0,Y 381.651,Z 280.288,A -85,B 0,C 180,E1 -12140.46,E2 -12140.46} C_VEL
LIN {X 0,Y 381.79,Z 278.673,A -85,B 0,C 180,E1 -12142.597,E2 -12142.597} C_VEL
LIN {X 0,Y 381.935,Z 277.271,A -85,B 0,C 180,E1 -12143.661,E2 -12143.661} C_VEL
LIN {X 0,Y 381.997,Z 274.357,A -85,B 0,C 180,E1 -12145.251,E2 -12145.251} C_VEL
LIN {X 0,Y 382.311,Z 270.401,A -85,B 0,C 180,E1 -12146.839,E2 -12146.839} C_VEL
LIN {X 0,Y 382.59,Z 265.328,A -85,B 0,C 180,E1 -12148.421,E2 -12148.421} C_VEL
LIN {X 0,Y 383.142,Z 258.925,A -85,B 0,C 180,E1 -12150,E2 -12150} C_VEL
LIN {X 0,Y 383.746,Z 250.972,A -85,B 0,C 180,E1 -12151.574,E2 -12151.574} C_VEL
LIN {X 0,Y 384.309,Z 242.879,A -85,B 0,C 180,E1 -12152.883,E2 -12152.883} C_VEL
LIN {X 0,Y 385.193,Z 234.021,A -85,B 0,C 180,E1 -12154.054,E2 -12154.054} C_VEL
LIN {X 0,Y 385.913,Z 224.501,A -85,B 0,C 180,E1 -12155.094,E2 -12155.094} C_VEL
LIN {X 0,Y 386.624,Z 214.27,A -85,B 0,C 180,E1 -12156,E2 -12156} C_VEL
LIN {X 0,Y 387.231,Z 202.103,A -85,B 0,C 180,E1 -12156.841,E2 -12156.841} C_VEL
LIN {X 0,Y 387.698,Z 188.593,A -85,B 0,C 180,E1 -12157.519,E2 -12157.519} C_VEL
LIN {X 0,Y 387.985,Z 178.01,A -85,B 0,C 180,E1 -12157.878,E2 -12157.878} C_VEL
LIN {X 0,Y 387.434,Z 172.237,A -85,B 0,C 180,E1 -12158.053,E2 -12158.053} C_VEL
LIN {X 0,Y 382.147,Z 153.496,A -85,B 0,C 180,E1 -12158.63,E2 -12158.63} C_VEL
LIN {X 0,Y 381.666,Z 147.672,A -85,B 0,C 180,E1 -12158.756,E2 -12158.756} C_VEL
LIN {X 0,Y 382.295,Z 90.506,A -85,B 0,C 180,E1 -12159.832,E2 -12159.832} C_VEL
LIN {X 0,Y 380.177,Z 80.542,A -85,B 0,C 180,E1 -12160.124,E2 -12160.124} C_VEL
LIN {X 0,Y 376.937,Z 70.435,A -85,B 0,C 180,E1 -12160.501,E2 -12160.501} C_VEL
LIN {X 0,Y 376.054,Z 65.638,A -85,B 0,C 180,E1 -12161.795,E2 -12161.795} C_VEL
LIN {X 0,Y 376.06,Z 65.639,A -85,B 0,C 180,E1 -12165.168,E2 -12165.168} C_VEL
LIN {X 0,Y 376.026,Z 65.648,A -85,B 0,C 180,E1 -12168.526,E2 -12168.526} C_VEL
LIN {X 0,Y 375.961,Z 65.653,A -85,B 0,C 180,E1 -12171.955,E2 -12171.955} C_VEL
LIN {X 0,Y 376.007,Z 65.645,A -85,B 0,C 180,E1 -12175.461,E2 -12175.461} C_VEL
LIN {X 0,Y 375.963,Z 65.65,A -85,B 0,C 180,E1 -12179.08,E2 -12179.08} C_VEL
LIN {X 0,Y 375.953,Z 65.651,A -85,B 0,C 180,E1 -12182.829,E2 -12182.829} C_VEL
LIN {X 0,Y 375.96,Z 65.653,A -85,B 0,C 180,E1 -12185.416,E2 -12185.416} C_VEL
LIN {X 0,Y 375.978,Z 65.649,A -85,B 0,C 180,E1 -12188.271,E2 -12188.271} C_VEL
LIN {X 0,Y 375.937,Z 65.66,A -85,B 0,C 180,E1 -12191.601,E2 -12191.601} C_VEL
LIN {X 0,Y 375.929,Z 65.658,A -85,B 0,C 180,E1 -12195.269,E2 -12195.269} C_VEL
LIN {X 0,Y 375.936,Z 65.653,A -85,B 0,C 180,E1 -12198.4,E2 -12198.4} C_VEL
LIN {X 0,Y 375.976,Z 65.65,A -85,B 0,C 180,E1 -12201.73,E2 -12201.73} C_VEL
LIN {X 0,Y 375.983,Z 65.651,A -85,B 0,C 180,E1 -12205.333,E2 -12205.333} C_VEL
LIN {X 0,Y 375.961,Z 65.652,A -85,B 0,C 180,E1 -12208.438,E2 -12208.438} C_VEL
LIN {X 0,Y 375.987,Z 65.648,A -85,B 0,C 180,E1 -12212.141,E2 -12212.141} C_VEL
LIN {X 0,Y 376.01,Z 65.648,A -85,B 0,C 180,E1 -12214.539,E2 -12214.539} C_VEL
LIN {X 0,Y 375.972,Z 65.65,A -85,B 0,C 180,E1 -12218.046,E2 -12218.046} C_VEL
LIN {X 0,Y 376.012,Z 65.644,A -85,B 0,C 180,E1 -12221.473,E2 -12221.473} C_VEL
LIN {X 0,Y 376.063,Z 65.64,A -85,B 0,C 180,E1 -12224.833,E2 -12224.833} C_VEL
LIN {X 0,Y 376.055,Z 65.643,A -85,B 0,C 180,E1 -12228.137,E2 -12228.137} C_VEL
LIN {X 0,Y 376.221,Z 65.622,A -85,B 0,C 180,E1 -12231.922,E2 -12231.922} C_VEL
LIN {X 0,Y 376.172,Z 65.625,A -85,B 0,C 180,E1 -12234.64,E2 -12234.64} C_VEL
LIN {X 0,Y 376.354,Z 65.607,A -85,B 0,C 180,E1 -12237.86,E2 -12237.86} C_VEL
LIN {X 0,Y 376.492,Z 65.589,A -85,B 0,C 180,E1 -12240,E2 -12240} C_VEL
LIN {X 0,Y 376.187,Z 65.624,A -85,B 0,C 180,E1 -12243.213,E2 -12243.213} C_VEL
LIN {X 0,Y 376.206,Z 65.62,A -85,B 0,C 180,E1 -12246.436,E2 -12246.436} C_VEL
LIN {X 0,Y 376.118,Z 65.635,A -85,B 0,C 180,E1 -12249.682,E2 -12249.682} C_VEL
LIN {X 0,Y 376.094,Z 65.637,A -85,B 0,C 180,E1 -12253.658,E2 -12253.658} C_VEL
LIN {X 0,Y 376.037,Z 65.645,A -85,B 0,C 180,E1 -12257.4,E2 -12257.4} C_VEL
LIN {X 0,Y 375.982,Z 65.651,A -85,B 0,C 180,E1 -12260.832,E2 -12260.832} C_VEL
LIN {X 0,Y 375.983,Z 65.648,A -85,B 0,C 180,E1 -12264.282,E2 -12264.282} C_VEL
LIN {X 0,Y 375.969,Z 65.653,A -85,B 0,C 180,E1 -12266.656,E2 -12266.656} C_VEL
LIN {X 0,Y 375.967,Z 65.652,A -85,B 0,C 180,E1 -12270.313,E2 -12270.313} C_VEL
LIN {X 0,Y 375.963,Z 65.651,A -85,B 0,C 180,E1 -12274.111,E2 -12274.111} C_VEL
LIN {X 0,Y 375.956,Z 65.655,A -85,B 0,C 180,E1 -12276.741,E2 -12276.741} C_VEL
LIN {X 0,Y 375.991,Z 65.649,A -85,B 0,C 180,E1 -12279.97,E2 -12279.97} C_VEL
LIN {X 0,Y 375.933,Z 65.655,A -85,B 0,C 180,E1 -12283.766,E2 -12283.766} C_VEL
LIN {X 0,Y 375.937,Z 65.654,A -85,B 0,C 180,E1 -12286.81,E2 -12286.81} C_VEL
LIN {X 0,Y 375.946,Z 65.654,A -85,B 0,C 180,E1 -12290.535,E2 -12290.535} C_VEL
LIN {X 0,Y 375.966,Z 65.652,A -85,B 0,C 180,E1 -12293.496,E2 -12293.496} C_VEL
LIN {X 0,Y 375.963,Z 65.656,A -85,B 0,C 180,E1 -12295.888,E2 -12295.888} C_VEL
LIN {X 0,Y 375.97,Z 65.656,A -85,B 0,C 180,E1 -12299.687,E2 -12299.687} C_VEL
LIN {X 0,Y 376.06,Z 65.77,A -85,B 0,C 180,E1 -12300.621,E2 -12300.621} C_VEL
LIN {X 0,Y 378.456,Z 77.443,A -85,B 0,C 180,E1 -12303.252,E2 -12303.252} C_VEL
LIN {X 0,Y 379.232,Z 83.095,A -85,B 0,C 180,E1 -12304.477,E2 -12304.477} C_VEL
LIN {X 0,Y 377.836,Z 101.207,A -85,B 0,C 180,E1 -12308.16,E2 -12308.16} C_VEL
LIN {X 0,Y 377.38,Z 108.006,A -85,B 0,C 180,E1 -12309.534,E2 -12309.534} C_VEL
LIN {X 0,Y 381.774,Z 143.112,A -85,B 0,C 180,E1 -12310.418,E2 -12310.418} C_VEL
LIN {X 0,Y 380.864,Z 216.843,A -85,B 0,C 180,E1 -12311.822,E2 -12311.822} C_VEL
LIN {X 0,Y 380.299,Z 230.193,A -85,B 0,C 180,E1 -12312.281,E2 -12312.281} C_VEL
LIN {X 0,Y 379.527,Z 242.413,A -85,B 0,C 180,E1 -12312.904,E2 -12312.904} C_VEL
LIN {X 0,Y 378.703,Z 253.932,A -85,B 0,C 180,E1 -12313.698,E2 -12313.698} C_VEL
LIN {X 0,Y 377.808,Z 265.765,A -85,B 0,C 180,E1 -12314.766,E2 -12314.766} C_VEL
LIN {X 0,Y 376.935,Z 276.381,A -85,B 0,C 180,E1 -12315.972,E2 -12315.972} C_VEL
LIN {X 0,Y 376.183,Z 285.943,A -85,B 0,C 180,E1 -12317.319,E2 -12317.319} C_VEL
LIN {X 0,Y 375.485,Z 295.141,A -85,B 0,C 180,E1 -12318.939,E2 -12318.939} C_VEL
LIN {X 0,Y 375.015,Z 302.549,A -85,B 0,C 180,E1 -12320.562,E2 -12320.562} C_VEL
LIN {X 0,Y 374.797,Z 307.566,A -85,B 0,C 180,E1 -12321.915,E2 -12321.915} C_VEL
LIN {X 0,Y 374.567,Z 312.421,A -85,B 0,C 180,E1 -12323.536,E2 -12323.536} C_VEL
LIN {X 0,Y 374.625,Z 316.147,A -85,B 0,C 180,E1 -12325.157,E2 -12325.157} C_VEL
LIN {X 0,Y 374.594,Z 318.827,A -85,B 0,C 180,E1 -12326.773,E2 -12326.773} C_VEL
LIN {X 0,Y 374.698,Z 320.092,A -85,B 0,C 180,E1 -12327.85,E2 -12327.85} C_VEL
LIN {X 0,Y 374.671,Z 320.938,A -85,B 0,C 180,E1 -12328.925,E2 -12328.925} C_VEL
LIN {X 0,Y 374.657,Z 321.345,A -85,B 0,C 180,E1 -12330,E2 -12330} C_VEL
LIN {X 0,Y 374.651,Z 321.358,A -85,B 0,C 180,E1 -12331.075,E2 -12331.075} C_VEL
LIN {X 0,Y 374.627,Z 320.984,A -85,B 0,C 180,E1 -12332.15,E2 -12332.15} C_VEL
LIN {X 0,Y 374.534,Z 320.214,A -85,B 0,C 180,E1 -12333.227,E2 -12333.227} C_VEL
LIN {X 0,Y 374.561,Z 319.009,A -85,B 0,C 180,E1 -12334.304,E2 -12334.304} C_VEL
LIN {X 0,Y 374.537,Z 316.29,A -85,B 0,C 180,E1 -12335.999,E2 -12335.999} C_VEL
LIN {X 0,Y 374.831,Z 311.436,A -85,B 0,C 180,E1 -12338.084,E2 -12338.084} C_VEL
LIN {X 0,Y 375.181,Z 306.397,A -85,B 0,C 180,E1 -12339.706,E2 -12339.706} C_VEL
LIN {X 0,Y 375.803,Z 300.097,A -85,B 0,C 180,E1 -12341.324,E2 -12341.324} C_VEL
LIN {X 0,Y 376.809,Z 292.248,A -85,B 0,C 180,E1 -12342.933,E2 -12342.933} C_VEL
LIN {X 0,Y 377.829,Z 282.566,A -85,B 0,C 180,E1 -12344.531,E2 -12344.531} C_VEL
LIN {X 0,Y 379.018,Z 272.406,A -85,B 0,C 180,E1 -12345.873,E2 -12345.873} C_VEL
LIN {X 0,Y 380.322,Z 261.019,A -85,B 0,C 180,E1 -12347.059,E2 -12347.059} C_VEL
LIN {X 0,Y 381.438,Z 249.877,A -85,B 0,C 180,E1 -12347.976,E2 -12347.976} C_VEL
LIN {X 0,Y 382.609,Z 237.438,A -85,B 0,C 180,E1 -12348.751,E2 -12348.751} C_VEL
LIN {X 0,Y 383.487,Z 225.089,A -85,B 0,C 180,E1 -12349.296,E2 -12349.296} C_VEL
LIN {X 0,Y 383.998,Z 211.34,A -85,B 0,C 180,E1 -12349.687,E2 -12349.687} C_VEL
LIN {X 0,Y 385.096,Z 142.908,A -85,B 0,C 180,E1 -12350.988,E2 -12350.988} C_VEL
LIN {X 0,Y 380.958,Z 117.444,A -85,B 0,C 180,E1 -12351.781,E2 -12351.781} C_VEL
LIN {X 0,Y 378.92,Z 107.252,A -85,B 0,C 180,E1 -12352.16,E2 -12352.16} C_VEL
LIN {X 0,Y 380.327,Z 92.972,A -85,B 0,C 180,E1 -12355.152,E2 -12355.152} C_VEL
LIN {X 0,Y 380.79,Z 87.613,A -85,B 0,C 180,E1 -12356.293,E2 -12356.293} C_VEL
LIN {X 0,Y 378.955,Z 78.216,A -85,B 0,C 180,E1 -12358.526,E2 -12358.526} C_VEL
LIN {X 0,Y 376.502,Z 67.917,A -85,B 0,C 180,E1 -12361.099,E2 -12361.099} C_VEL
LIN {X 0,Y 375.968,Z 65.652,A -85,B 0,C 180,E1 -12361.718,E2 -12361.718} C_VEL
LIN {X 0,Y 375.96,Z 65.653,A -85,B 0,C 180,E1 -12365.415,E2 -12365.415} C_VEL
LIN {X 0,Y 375.976,Z 65.648,A -85,B 0,C 180,E1 -12368.27,E2 -12368.27} C_VEL
LIN {X 0,Y 375.937,Z 65.658,A -85,B 0,C 180,E1 -12371.601,E2 -12371.601} C_VEL
LIN {X 0,Y 375.93,Z 65.652,A -85,B 0,C 180,E1 -12375.269,E2 -12375.269} C_VEL
LIN {X 0,Y 375.937,Z 65.651,A -85,B 0,C 180,E1 -12378.399,E2 -12378.399} C_VEL
LIN {X 0,Y 375.975,Z 65.649,A -85,B 0,C 180,E1 -12381.73,E2 -12381.73} C_VEL
LIN {X 0,Y 375.982,Z 65.649,A -85,B 0,C 180,E1 -12385.333,E2 -12385.333} C_VEL
LIN {X 0,Y 375.961,Z 65.652,A -85,B 0,C 180,E1 -12388.438,E2 -12388.438} C_VEL
LIN {X 0,Y 375.999,Z 65.647,A -85,B 0,C 180,E1 -12392.141,E2 -12392.141} C_VEL
LIN {X 0,Y 376.009,Z 65.642,A -85,B 0,C 180,E1 -12394.539,E2 -12394.539} C_VEL
LIN {X 0,Y 375.967,Z 65.647,A -85,B 0,C 180,E1 -12398.046,E2 -12398.046} C_VEL
LIN {X 0,Y 376.012,Z 65.644,A -85,B 0,C 180,E1 -12401.473,E2 -12401.473} C_VEL
LIN {X 0,Y 376.062,Z 65.641,A -85,B 0,C 180,E1 -12404.833,E2 -12404.833} C_VEL
LIN {X 0,Y 376.053,Z 65.635,A -85,B 0,C 180,E1 -12408.137,E2 -12408.137} C_VEL
LIN {X 0,Y 376.222,Z 65.619,A -85,B 0,C 180,E1 -12411.919,E2 -12411.919} C_VEL
LIN {X 0,Y 376.172,Z 65.626,A -85,B 0,C 180,E1 -12414.64,E2 -12414.64} C_VEL
LIN {X 0,Y 376.353,Z 65.598,A -85,B 0,C 180,E1 -12417.859,E2 -12417.859} C_VEL
LIN {X 0,Y 376.491,Z 65.587,A -85,B 0,C 180,E1 -12420,E2 -12420} C_VEL
LIN {X 0,Y 376.186,Z 65.62,A -85,B 0,C 180,E1 -12423.213,E2 -12423.213} C_VEL
LIN {X 0,Y 376.216,Z 65.619,A -85,B 0,C 180,E1 -12426.581,E2 -12426.581} C_VEL
LIN {X 0,Y 376.116,Z 65.63,A -85,B 0,C 180,E1 -12429.681,E2 -12429.681} C_VEL
LIN {X 0,Y 376.092,Z 65.629,A -85,B 0,C 180,E1 -12433.657,E2 -12433.657} C_VEL
LIN {X 0,Y 376.035,Z 65.641,A -85,B 0,C 180,E1 -12437.4,E2 -12437.4} C_VEL
LIN {X 0,Y 375.981,Z 65.653,A -85,B 0,C 180,E1 -12440.832,E2 -12440.832} C_VEL
LIN {X 0,Y 375.987,Z 65.647,A -85,B 0,C 180,E1 -12444.282,E2 -12444.282} C_VEL
LIN {X 0,Y 375.968,Z 65.65,A -85,B 0,C 180,E1 -12446.656,E2 -12446.656} C_VEL
LIN {X 0,Y 375.965,Z 65.652,A -85,B 0,C 180,E1 -12450.313,E2 -12450.313} C_VEL
LIN {X 0,Y 375.962,Z 65.651,A -85,B 0,C 180,E1 -12454.111,E2 -12454.111} C_VEL
LIN {X 0,Y 375.954,Z 65.652,A -85,B 0,C 180,E1 -12456.741,E2 -12456.741} C_VEL
LIN {X 0,Y 375.97,Z 65.645,A -85,B 0,C 180,E1 -12459.967,E2 -12459.967} C_VEL
LIN {X 0,Y 375.931,Z 65.661,A -85,B 0,C 180,E1 -12463.766,E2 -12463.766} C_VEL
LIN {X 0,Y 375.935,Z 65.657,A -85,B 0,C 180,E1 -12466.81,E2 -12466.81} C_VEL
LIN {X 0,Y 375.944,Z 65.655,A -85,B 0,C 180,E1 -12470.535,E2 -12470.535} C_VEL
LIN {X 0,Y 375.963,Z 65.656,A -85,B 0,C 180,E1 -12473.496,E2 -12473.496} C_VEL
LIN {X 0,Y 376.007,Z 65.78,A -85,B 0,C 180,E1 -12476.176,E2 -12476.176} C_VEL
LIN {X 0,Y 377.216,Z 71.252,A -85,B 0,C 180,E1 -12477.79,E2 -12477.79} C_VEL
LIN {X 0,Y 385.284,Z 90.803,A -85,B 0,C 180,E1 -12478.765,E2 -12478.765} C_VEL
LIN {X 0,Y 386.017,Z 94.363,A -85,B 0,C 180,E1 -12478.888,E2 -12478.888} C_VEL
LIN {X 0,Y 384.358,Z 178.175,A -85,B 0,C 180,E1 -12480.491,E2 -12480.491} C_VEL
LIN {X 0,Y 383.891,Z 191.649,A -85,B 0,C 180,E1 -12480.978,E2 -12480.978} C_VEL
LIN {X 0,Y 383.284,Z 204.285,A -85,B 0,C 180,E1 -12481.659,E2 -12481.659} C_VEL
LIN {X 0,Y 382.368,Z 216.109,A -85,B 0,C 180,E1 -12482.52,E2 -12482.52} C_VEL
LIN {X 0,Y 381.221,Z 227.574,A -85,B 0,C 180,E1 -12483.592,E2 -12483.592} C_VEL
LIN {X 0,Y 380.11,Z 238.061,A -85,B 0,C 180,E1 -12484.833,E2 -12484.833} C_VEL
LIN {X 0,Y 379.005,Z 247.392,A -85,B 0,C 180,E1 -12486.214,E2 -12486.214} C_VEL
LIN {X 0,Y 377.872,Z 256.417,A -85,B 0,C 180,E1 -12487.875,E2 -12487.875} C_VEL
LIN {X 0,Y 376.925,Z 263.574,A -85,B 0,C 180,E1 -12489.537,E2 -12489.537} C_VEL
LIN {X 0,Y 376.078,Z 270.045,A -85,B 0,C 180,E1 -12491.477,E2 -12491.477} C_VEL
LIN {X 0,Y 375.542,Z 274.257,A -85,B 0,C 180,E1 -12493.138,E2 -12493.138} C_VEL
LIN {X 0,Y 375.143,Z 277.363,A -85,B 0,C 180,E1 -12494.795,E2 -12494.795} C_VEL
LIN {X 0,Y 374.912,Z 278.89,A -85,B 0,C 180,E1 -12495.895,E2 -12495.895} C_VEL
LIN {X 0,Y 374.795,Z 280.08,A -85,B 0,C 180,E1 -12497.183,E2 -12497.183} C_VEL
LIN {X 0,Y 374.609,Z 280.867,A -85,B 0,C 180,E1 -12499.187,E2 -12499.187} C_VEL
LIN {X 0,Y 374.557,Z 280.733,A -85,B 0,C 180,E1 -12500.278,E2 -12500.278} C_VEL
LIN {X 0,Y 374.606,Z 280.159,A -85,B 0,C 180,E1 -12501.368,E2 -12501.368} C_VEL
LIN {X 0,Y 374.863,Z 277.839,A -85,B 0,C 180,E1 -12503.541,E2 -12503.541} C_VEL
LIN {X 0,Y 374.917,Z 275,A -85,B 0,C 180,E1 -12505.161,E2 -12505.161} C_VEL
LIN {X 0,Y 375.226,Z 271.131,A -85,B 0,C 180,E1 -12506.779,E2 -12506.779} C_VEL
LIN {X 0,Y 375.492,Z 266.158,A -85,B 0,C 180,E1 -12508.391,E2 -12508.391} C_VEL
LIN {X 0,Y 376.049,Z 259.897,A -85,B 0,C 180,E1 -12510,E2 -12510} C_VEL
LIN {X 0,Y 376.686,Z 252.072,A -85,B 0,C 180,E1 -12511.604,E2 -12511.604} C_VEL
LIN {X 0,Y 377.264,Z 244.122,A -85,B 0,C 180,E1 -12512.937,E2 -12512.937} C_VEL
LIN {X 0,Y 378.08,Z 235.453,A -85,B 0,C 180,E1 -12514.131,E2 -12514.131} C_VEL
LIN {X 0,Y 378.993,Z 224.849,A -85,B 0,C 180,E1 -12515.32,E2 -12515.32} C_VEL
LIN {X 0,Y 379.732,Z 214.608,A -85,B 0,C 180,E1 -12516.242,E2 -12516.242} C_VEL
LIN {X 0,Y 380.365,Z 202.42,A -85,B 0,C 180,E1 -12517.098,E2 -12517.098} C_VEL
LIN {X 0,Y 380.853,Z 188.885,A -85,B 0,C 180,E1 -12517.789,E2 -12517.789} C_VEL
LIN {X 0,Y 381.233,Z 175.928,A -85,B 0,C 180,E1 -12518.214,E2 -12518.214} C_VEL
LIN {X 0,Y 381.666,Z 147.672,A -85,B 0,C 180,E1 -12518.756,E2 -12518.756} C_VEL
LIN {X 0,Y 381.195,Z 141.858,A -85,B 0,C 180,E1 -12518.889,E2 -12518.889} C_VEL
LIN {X 0,Y 375.913,Z 123.137,A -85,B 0,C 180,E1 -12519.489,E2 -12519.489} C_VEL
LIN {X 0,Y 375.275,Z 117.323,A -85,B 0,C 180,E1 -12519.632,E2 -12519.632} C_VEL
LIN {X 0,Y 375.488,Z 91.36,A -85,B 0,C 180,E1 -12520.134,E2 -12520.134} C_VEL
LIN {X 0,Y 373.394,Z 81.768,A -85,B 0,C 180,E1 -12520.424,E2 -12520.424} C_VEL
LIN {X 0,Y 369.827,Z 70.835,A -85,B 0,C 180,E1 -12520.834,E2 -12520.834} C_VEL
LIN {X 0,Y 369.019,Z 66.516,A -85,B 0,C 180,E1 -12522.023,E2 -12522.023} C_VEL
LIN {X 0,Y 369,Z 66.517,A -85,B 0,C 180,E1 -12525.465,E2 -12525.465} C_VEL
LIN {X 0,Y 368.985,Z 66.521,A -85,B 0,C 180,E1 -12528.893,E2 -12528.893} C_VEL
LIN {X 0,Y 368.927,Z 66.532,A -85,B 0,C 180,E1 -12532.396,E2 -12532.396} C_VEL
LIN {X 0,Y 369.001,Z 66.522,A -85,B 0,C 180,E1 -12535.98,E2 -12535.98} C_VEL
LIN {X 0,Y 368.916,Z 66.531,A -85,B 0,C 180,E1 -12539.691,E2 -12539.691} C_VEL
LIN {X 0,Y 368.9,Z 66.53,A -85,B 0,C 180,E1 -12543.044,E2 -12543.044} C_VEL
LIN {X 0,Y 368.92,Z 66.53,A -85,B 0,C 180,E1 -12546.197,E2 -12546.197} C_VEL
LIN {X 0,Y 368.907,Z 66.529,A -85,B 0,C 180,E1 -12548.953,E2 -12548.953} C_VEL
LIN {X 0,Y 368.884,Z 66.534,A -85,B 0,C 180,E1 -12552.01,E2 -12552.01} C_VEL
LIN {X 0,Y 368.882,Z 66.535,A -85,B 0,C 180,E1 -12555.176,E2 -12555.176} C_VEL
LIN {X 0,Y 368.885,Z 66.532,A -85,B 0,C 180,E1 -12558.178,E2 -12558.178} C_VEL
LIN {X 0,Y 368.911,Z 66.534,A -85,B 0,C 180,E1 -12561.36,E2 -12561.36} C_VEL
LIN {X 0,Y 368.939,Z 66.531,A -85,B 0,C 180,E1 -12565.147,E2 -12565.147} C_VEL
LIN {X 0,Y 368.932,Z 66.531,A -85,B 0,C 180,E1 -12569.047,E2 -12569.047} C_VEL
LIN {X 0,Y 368.966,Z 66.528,A -85,B 0,C 180,E1 -12572.797,E2 -12572.797} C_VEL
LIN {X 0,Y 368.949,Z 66.525,A -85,B 0,C 180,E1 -12576.113,E2 -12576.113} C_VEL
LIN {X 0,Y 368.94,Z 66.526,A -85,B 0,C 180,E1 -12579.947,E2 -12579.947} C_VEL
LIN {X 0,Y 368.98,Z 66.52,A -85,B 0,C 180,E1 -12583.399,E2 -12583.399} C_VEL
LIN {X 0,Y 369.062,Z 66.512,A -85,B 0,C 180,E1 -12586.79,E2 -12586.79} C_VEL
LIN {X 0,Y 369.069,Z 66.514,A -85,B 0,C 180,E1 -12590.132,E2 -12590.132} C_VEL
LIN {X 0,Y 369.199,Z 66.493,A -85,B 0,C 180,E1 -12593.442,E2 -12593.442} C_VEL
LIN {X 0,Y 369.319,Z 66.483,A -85,B 0,C 180,E1 -12597.819,E2 -12597.819} C_VEL
LIN {X 0,Y 369.462,Z 66.465,A -85,B 0,C 180,E1 -12600,E2 -12600} C_VEL
LIN {X 0,Y 369.321,Z 66.48,A -85,B 0,C 180,E1 -12602.181,E2 -12602.181} C_VEL
LIN {X 0,Y 369.166,Z 66.497,A -85,B 0,C 180,E1 -12606.559,E2 -12606.559} C_VEL
LIN {X 0,Y 369.068,Z 66.511,A -85,B 0,C 180,E1 -12609.868,E2 -12609.868} C_VEL
LIN {X 0,Y 369.042,Z 66.514,A -85,B 0,C 180,E1 -12613.772,E2 -12613.772} C_VEL
LIN {X 0,Y 368.995,Z 66.519,A -85,B 0,C 180,E1 -12617.743,E2 -12617.743} C_VEL
LIN {X 0,Y 368.932,Z 66.531,A -85,B 0,C 180,E1 -12621.22,E2 -12621.22} C_VEL
LIN {X 0,Y 368.943,Z 66.529,A -85,B 0,C 180,E1 -12624.777,E2 -12624.777} C_VEL
LIN {X 0,Y 368.934,Z 66.528,A -85,B 0,C 180,E1 -12628.44,E2 -12628.44} C_VEL
LIN {X 0,Y 368.914,Z 66.532,A -85,B 0,C 180,E1 -12630.987,E2 -12630.987} C_VEL
LIN {X 0,Y 368.94,Z 66.528,A -85,B 0,C 180,E1 -12634.853,E2 -12634.853} C_VEL
LIN {X 0,Y 368.911,Z 66.533,A -85,B 0,C 180,E1 -12638.64,E2 -12638.64} C_VEL
LIN {X 0,Y 368.885,Z 66.535,A -85,B 0,C 180,E1 -12642.009,E2 -12642.009} C_VEL
LIN {X 0,Y 368.883,Z 66.532,A -85,B 0,C 180,E1 -12645.176,E2 -12645.176} C_VEL
LIN {X 0,Y 368.877,Z 66.538,A -85,B 0,C 180,E1 -12648.176,E2 -12648.176} C_VEL
LIN {X 0,Y 368.883,Z 66.533,A -85,B 0,C 180,E1 -12651.365,E2 -12651.365} C_VEL
LIN {X 0,Y 368.939,Z 66.525,A -85,B 0,C 180,E1 -12655.146,E2 -12655.146} C_VEL
LIN {X 0,Y 368.932,Z 66.527,A -85,B 0,C 180,E1 -12659.046,E2 -12659.046} C_VEL
LIN {X 0,Y 368.974,Z 66.696,A -85,B 0,C 180,E1 -12660.371,E2 -12660.371} C_VEL
LIN {X 0,Y 371.64,Z 79.488,A -85,B 0,C 180,E1 -12663.312,E2 -12663.312} C_VEL
LIN {X 0,Y 372.23,Z 84.939,A -85,B 0,C 180,E1 -12664.507,E2 -12664.507} C_VEL
LIN {X 0,Y 370.742,Z 103.065,A -85,B 0,C 180,E1 -12668.26,E2 -12668.26} C_VEL
LIN {X 0,Y 370.431,Z 107.648,A -85,B 0,C 180,E1 -12669.205,E2 -12669.205} C_VEL
LIN {X 0,Y 374.963,Z 144.234,A -85,B 0,C 180,E1 -12670.14,E2 -12670.14} C_VEL
LIN {X 0,Y 373.992,Z 216.745,A -85,B 0,C 180,E1 -12671.547,E2 -12671.547} C_VEL
LIN {X 0,Y 373.417,Z 230.004,A -85,B 0,C 180,E1 -12672.014,E2 -12672.014} C_VEL
LIN {X 0,Y 372.635,Z 242.178,A -85,B 0,C 180,E1 -12672.649,E2 -12672.649} C_VEL
LIN {X 0,Y 371.711,Z 254.467,A -85,B 0,C 180,E1 -12673.524,E2 -12673.524} C_VEL
LIN {X 0,Y 370.806,Z 266.124,A -85,B 0,C 180,E1 -12674.612,E2 -12674.612} C_VEL
LIN {X 0,Y 369.888,Z 276.687,A -85,B 0,C 180,E1 -12675.849,E2 -12675.849} C_VEL
LIN {X 0,Y 369.204,Z 285.189,A -85,B 0,C 180,E1 -12677.075,E2 -12677.075} C_VEL
LIN {X 0,Y 368.618,Z 293.091,A -85,B 0,C 180,E1 -12678.452,E2 -12678.452} C_VEL
LIN {X 0,Y 368.052,Z 300.793,A -85,B 0,C 180,E1 -12680.104,E2 -12680.104} C_VEL
LIN {X 0,Y 367.731,Z 306.986,A -85,B 0,C 180,E1 -12681.759,E2 -12681.759} C_VEL
LIN {X 0,Y 367.491,Z 311.884,A -85,B 0,C 180,E1 -12683.411,E2 -12683.411} C_VEL
LIN {X 0,Y 367.529,Z 315.649,A -85,B 0,C 180,E1 -12685.063,E2 -12685.063} C_VEL
LIN {X 0,Y 367.503,Z 318.365,A -85,B 0,C 180,E1 -12686.711,E2 -12686.711} C_VEL
LIN {X 0,Y 367.614,Z 319.648,A -85,B 0,C 180,E1 -12687.809,E2 -12687.809} C_VEL
LIN {X 0,Y 367.605,Z 320.521,A -85,B 0,C 180,E1 -12688.904,E2 -12688.904} C_VEL
LIN {X 0,Y 367.588,Z 320.952,A -85,B 0,C 180,E1 -12690,E2 -12690} C_VEL
LIN {X 0,Y 367.584,Z 320.983,A -85,B 0,C 180,E1 -12691.095,E2 -12691.095} C_VEL
LIN {X 0,Y 367.527,Z 320.623,A -85,B 0,C 180,E1 -12692.192,E2 -12692.192} C_VEL
LIN {X 0,Y 367.446,Z 319.874,A -85,B 0,C 180,E1 -12693.289,E2 -12693.289} C_VEL
LIN {X 0,Y 367.462,Z 318.698,A -85,B 0,C 180,E1 -12694.388,E2 -12694.388} C_VEL
LIN {X 0,Y 367.458,Z 316.273,A -85,B 0,C 180,E1 -12695.981,E2 -12695.981} C_VEL
LIN {X 0,Y 367.663,Z 312.635,A -85,B 0,C 180,E1 -12697.69,E2 -12697.69} C_VEL
LIN {X 0,Y 367.983,Z 308.022,A -85,B 0,C 180,E1 -12699.343,E2 -12699.343} C_VEL
LIN {X 0,Y 368.685,Z 301.073,A -85,B 0,C 180,E1 -12701.267,E2 -12701.267} C_VEL
LIN {X 0,Y 369.68,Z 293.583,A -85,B 0,C 180,E1 -12702.908,E2 -12702.908} C_VEL
LIN {X 0,Y 370.695,Z 284.619,A -85,B 0,C 180,E1 -12704.494,E2 -12704.494} C_VEL
LIN {X 0,Y 371.903,Z 274.647,A -85,B 0,C 180,E1 -12705.903,E2 -12705.903} C_VEL
LIN {X 0,Y 373.218,Z 263.997,A -85,B 0,C 180,E1 -12707.112,E2 -12707.112} C_VEL
LIN {X 0,Y 374.391,Z 253.72,A -85,B 0,C 180,E1 -12708.043,E2 -12708.043} C_VEL
LIN {X 0,Y 375.544,Z 241.494,A -85,B 0,C 180,E1 -12708.904,E2 -12708.904} C_VEL
LIN {X 0,Y 376.696,Z 227.9,A -85,B 0,C 180,E1 -12709.587,E2 -12709.587} C_VEL
LIN {X 0,Y 377.296,Z 215.13,A -85,B 0,C 180,E1 -12710.016,E2 -12710.016} C_VEL
LIN {X 0,Y 378.676,Z 144.606,A -85,B 0,C 180,E1 -12711.383,E2 -12711.383} C_VEL
LIN {X 0,Y 375.227,Z 122.534,A -85,B 0,C 180,E1 -12712.078,E2 -12712.078} C_VEL
LIN {X 0,Y 372.16,Z 106.962,A -85,B 0,C 180,E1 -12712.631,E2 -12712.631} C_VEL
LIN {X 0,Y 373.917,Z 90.225,A -85,B 0,C 180,E1 -12716.212,E2 -12716.212} C_VEL
LIN {X 0,Y 373.199,Z 84.894,A -85,B 0,C 180,E1 -12717.471,E2 -12717.471} C_VEL
LIN {X 0,Y 370.48,Z 72.814,A -85,B 0,C 180,E1 -12720.494,E2 -12720.494} C_VEL
LIN {X 0,Y 368.942,Z 66.53,A -85,B 0,C 180,E1 -12722.16,E2 -12722.16} C_VEL
LIN {X 0,Y 368.931,Z 66.529,A -85,B 0,C 180,E1 -12725.001,E2 -12725.001} C_VEL
LIN {X 0,Y 368.91,Z 66.525,A -85,B 0,C 180,E1 -12728.64,E2 -12728.64} C_VEL
LIN {X 0,Y 368.884,Z 66.532,A -85,B 0,C 180,E1 -12732.009,E2 -12732.009} C_VEL
LIN {X 0,Y 368.882,Z 66.529,A -85,B 0,C 180,E1 -12735.176,E2 -12735.176} C_VEL
LIN {X 0,Y 368.885,Z 66.531,A -85,B 0,C 180,E1 -12738.178,E2 -12738.178} C_VEL
LIN {X 0,Y 368.91,Z 66.529,A -85,B 0,C 180,E1 -12741.36,E2 -12741.36} C_VEL
LIN {X 0,Y 368.939,Z 66.529,A -85,B 0,C 180,E1 -12745.147,E2 -12745.147} C_VEL
LIN {X 0,Y 368.932,Z 66.529,A -85,B 0,C 180,E1 -12749.047,E2 -12749.047} C_VEL
LIN {X 0,Y 368.983,Z 66.522,A -85,B 0,C 180,E1 -12751.564,E2 -12751.564} C_VEL
LIN {X 0,Y 369.003,Z 66.513,A -85,B 0,C 180,E1 -12754.02,E2 -12754.02} C_VEL
LIN {X 0,Y 368.936,Z 66.523,A -85,B 0,C 180,E1 -12757.605,E2 -12757.605} C_VEL
LIN {X 0,Y 368.962,Z 66.523,A -85,B 0,C 180,E1 -12761.106,E2 -12761.106} C_VEL
LIN {X 0,Y 369.002,Z 66.52,A -85,B 0,C 180,E1 -12764.535,E2 -12764.535} C_VEL
LIN {X 0,Y 369.009,Z 66.511,A -85,B 0,C 180,E1 -12767.907,E2 -12767.907} C_VEL
LIN {X 0,Y 369.169,Z 66.498,A -85,B 0,C 180,E1 -12771.869,E2 -12771.869} C_VEL
LIN {X 0,Y 369.145,Z 66.502,A -85,B 0,C 180,E1 -12774.537,E2 -12774.537} C_VEL
LIN {X 0,Y 369.318,Z 66.474,A -85,B 0,C 180,E1 -12777.819,E2 -12777.819} C_VEL
LIN {X 0,Y 369.46,Z 66.463,A -85,B 0,C 180,E1 -12780,E2 -12780} C_VEL
LIN {X 0,Y 369.32,Z 66.477,A -85,B 0,C 180,E1 -12782.181,E2 -12782.181} C_VEL
LIN {X 0,Y 369.189,Z 66.495,A -85,B 0,C 180,E1 -12786.564,E2 -12786.564} C_VEL
LIN {X 0,Y 369.067,Z 66.51,A -85,B 0,C 180,E1 -12789.868,E2 -12789.868} C_VEL
LIN {X 0,Y 369.04,Z 66.507,A -85,B 0,C 180,E1 -12793.772,E2 -12793.772} C_VEL
LIN {X 0,Y 368.993,Z 66.516,A -85,B 0,C 180,E1 -12797.743,E2 -12797.743} C_VEL
LIN {X 0,Y 368.932,Z 66.529,A -85,B 0,C 180,E1 -12801.219,E2 -12801.219} C_VEL
LIN {X 0,Y 368.945,Z 66.529,A -85,B 0,C 180,E1 -12804.776,E2 -12804.776} C_VEL
LIN {X 0,Y 368.933,Z 66.528,A -85,B 0,C 180,E1 -12808.44,E2 -12808.44} C_VEL
LIN {X 0,Y 368.912,Z 66.529,A -85,B 0,C 180,E1 -12810.987,E2 -12810.987} C_VEL
LIN {X 0,Y 368.938,Z 66.529,A -85,B 0,C 180,E1 -12814.853,E2 -12814.853} C_VEL
LIN {X 0,Y 368.881,Z 66.536,A -85,B 0,C 180,E1 -12818.634,E2 -12818.634} C_VEL
LIN {X 0,Y 368.875,Z 66.529,A -85,B 0,C 180,E1 -12822.008,E2 -12822.008} C_VEL
LIN {X 0,Y 368.881,Z 66.537,A -85,B 0,C 180,E1 -12825.176,E2 -12825.176} C_VEL
LIN {X 0,Y 368.882,Z 66.537,A -85,B 0,C 180,E1 -12828.177,E2 -12828.177} C_VEL
LIN {X 0,Y 368.88,Z 66.537,A -85,B 0,C 180,E1 -12831.365,E2 -12831.365} C_VEL
LIN {X 0,Y 368.937,Z 66.534,A -85,B 0,C 180,E1 -12835.146,E2 -12835.146} C_VEL
LIN {X 0,Y 368.946,Z 66.585,A -85,B 0,C 180,E1 -12835.727,E2 -12835.727} C_VEL
LIN {X 0,Y 370.125,Z 71.691,A -85,B 0,C 180,E1 -12837.264,E2 -12837.264} C_VEL
LIN {X 0,Y 379.053,Z 93,A -85,B 0,C 180,E1 -12838.373,E2 -12838.373} C_VEL
LIN {X 0,Y 379.576,Z 95.665,A -85,B 0,C 180,E1 -12838.465,E2 -12838.465} C_VEL
LIN {X 0,Y 377.832,Z 178.815,A -85,B 0,C 180,E1 -12840.083,E2 -12840.083} C_VEL
LIN {X 0,Y 377.333,Z 192.202,A -85,B 0,C 180,E1 -12840.577,E2 -12840.577} C_VEL
LIN {X 0,Y 376.711,Z 204.681,A -85,B 0,C 180,E1 -12841.264,E2 -12841.264} C_VEL
LIN {X 0,Y 375.777,Z 216.323,A -85,B 0,C 180,E1 -12842.124,E2 -12842.124} C_VEL
LIN {X 0,Y 374.542,Z 228.026,A -85,B 0,C 180,E1 -12843.234,E2 -12843.234} C_VEL
LIN {X 0,Y 373.357,Z 238.664,A -85,B 0,C 180,E1 -12844.52,E2 -12844.52} C_VEL
LIN {X 0,Y 372.313,Z 246.982,A -85,B 0,C 180,E1 -12845.759,E2 -12845.759} C_VEL
LIN {X 0,Y 371.111,Z 256.14,A -85,B 0,C 180,E1 -12847.45,E2 -12847.45} C_VEL
LIN {X 0,Y 370.094,Z 263.455,A -85,B 0,C 180,E1 -12849.142,E2 -12849.142} C_VEL
LIN {X 0,Y 369.396,Z 268.346,A -85,B 0,C 180,E1 -12850.552,E2 -12850.552} C_VEL
LIN {X 0,Y 368.736,Z 273.339,A -85,B 0,C 180,E1 -12852.361,E2 -12852.361} C_VEL
LIN {X 0,Y 368.252,Z 276.605,A -85,B 0,C 180,E1 -12853.935,E2 -12853.935} C_VEL
LIN {X 0,Y 367.877,Z 279.106,A -85,B 0,C 180,E1 -12855.62,E2 -12855.62} C_VEL
LIN {X 0,Y 367.744,Z 280.47,A -85,B 0,C 180,E1 -12857.076,E2 -12857.076} C_VEL
LIN {X 0,Y 367.529,Z 281.235,A -85,B 0,C 180,E1 -12858.976,E2 -12858.976} C_VEL
LIN {X 0,Y 367.468,Z 281.153,A -85,B 0,C 180,E1 -12860.088,E2 -12860.088} C_VEL
LIN {X 0,Y 367.504,Z 280.645,A -85,B 0,C 180,E1 -12861.2,E2 -12861.2} C_VEL
LIN {X 0,Y 367.74,Z 278.402,A -85,B 0,C 180,E1 -12863.416,E2 -12863.416} C_VEL
LIN {X 0,Y 367.841,Z 275.64,A -85,B 0,C 180,E1 -12865.068,E2 -12865.068} C_VEL
LIN {X 0,Y 368.142,Z 271.857,A -85,B 0,C 180,E1 -12866.717,E2 -12866.717} C_VEL
LIN {X 0,Y 368.398,Z 266.978,A -85,B 0,C 180,E1 -12868.36,E2 -12868.36} C_VEL
LIN {X 0,Y 368.957,Z 260.823,A -85,B 0,C 180,E1 -12870,E2 -12870} C_VEL
LIN {X 0,Y 369.63,Z 253.165,A -85,B 0,C 180,E1 -12871.634,E2 -12871.634} C_VEL
LIN {X 0,Y 370.386,Z 243.585,A -85,B 0,C 180,E1 -12873.263,E2 -12873.263} C_VEL
LIN {X 0,Y 371.31,Z 234.717,A -85,B 0,C 180,E1 -12874.478,E2 -12874.478} C_VEL
LIN {X 0,Y 372.086,Z 225.18,A -85,B 0,C 180,E1 -12875.555,E2 -12875.555} C_VEL
LIN {X 0,Y 372.846,Z 214.929,A -85,B 0,C 180,E1 -12876.494,E2 -12876.494} C_VEL
LIN {X 0,Y 373.506,Z 202.716,A -85,B 0,C 180,E1 -12877.365,E2 -12877.365} C_VEL
LIN {X 0,Y 373.991,Z 189.903,A -85,B 0,C 180,E1 -12878.034,E2 -12878.034} C_VEL
LIN {X 0,Y 374.347,Z 177.475,A -85,B 0,C 180,E1 -12878.468,E2 -12878.468} C_VEL
LIN {X 0,Y 375.275,Z 117.323,A -85,B 0,C 180,E1 -12879.632,E2 -12879.632} C_VEL
LIN {X 0,Y 374.75,Z 111.504,A -85,B 0,C 180,E1 -12879.771,E2 -12879.771} C_VEL
LIN {X 0,Y 372.324,Z 102.114,A -85,B 0,C 180,E1 -12880.072,E2 -12880.072} C_VEL
LIN {X 0,Y 367.749,Z 87.16,A -85,B 0,C 180,E1 -12880.594,E2 -12880.594} C_VEL
LIN {X 0,Y 362.668,Z 71.151,A -85,B 0,C 180,E1 -12881.209,E2 -12881.209} C_VEL
LIN {X 0,Y 361.985,Z 67.393,A -85,B 0,C 180,E1 -12882.261,E2 -12882.261} C_VEL
LIN {X 0,Y 361.963,Z 67.4,A -85,B 0,C 180,E1 -12884.621,E2 -12884.621} C_VEL
LIN {X 0,Y 361.961,Z 67.397,A -85,B 0,C 180,E1 -12888.099,E2 -12888.099} C_VEL
LIN {X 0,Y 361.864,Z 67.407,A -85,B 0,C 180,E1 -12891.655,E2 -12891.655} C_VEL
LIN {X 0,Y 361.928,Z 67.398,A -85,B 0,C 180,E1 -12895.29,E2 -12895.29} C_VEL
LIN {X 0,Y 361.914,Z 67.403,A -85,B 0,C 180,E1 -12897.779,E2 -12897.779} C_VEL
LIN {X 0,Y 361.84,Z 67.412,A -85,B 0,C 180,E1 -12901.63,E2 -12901.63} C_VEL
LIN {X 0,Y 361.876,Z 67.407,A -85,B 0,C 180,E1 -12905.345,E2 -12905.345} C_VEL
LIN {X 0,Y 361.873,Z 67.406,A -85,B 0,C 180,E1 -12909.027,E2 -12909.027} C_VEL
LIN {X 0,Y 361.838,Z 67.41,A -85,B 0,C 180,E1 -12912.829,E2 -12912.829} C_VEL
LIN {X 0,Y 361.82,Z 67.413,A -85,B 0,C 180,E1 -12915.947,E2 -12915.947} C_VEL
LIN {X 0,Y 361.838,Z 67.415,A -85,B 0,C 180,E1 -12919.245,E2 -12919.245} C_VEL
LIN {X 0,Y 361.866,Z 67.408,A -85,B 0,C 180,E1 -12922.777,E2 -12922.777} C_VEL
LIN {X 0,Y 361.857,Z 67.408,A -85,B 0,C 180,E1 -12925.72,E2 -12925.72} C_VEL
LIN {X 0,Y 361.876,Z 67.405,A -85,B 0,C 180,E1 -12929.672,E2 -12929.672} C_VEL
LIN {X 0,Y 361.957,Z 67.395,A -85,B 0,C 180,E1 -12933.475,E2 -12933.475} C_VEL
LIN {X 0,Y 361.896,Z 67.404,A -85,B 0,C 180,E1 -12937.145,E2 -12937.145} C_VEL
LIN {X 0,Y 361.91,Z 67.405,A -85,B 0,C 180,E1 -12940.724,E2 -12940.724} C_VEL
LIN {X 0,Y 361.937,Z 67.398,A -85,B 0,C 180,E1 -12943.066,E2 -12943.066} C_VEL
LIN {X 0,Y 362.003,Z 67.393,A -85,B 0,C 180,E1 -12946.528,E2 -12946.528} C_VEL
LIN {X 0,Y 362.006,Z 67.392,A -85,B 0,C 180,E1 -12949.937,E2 -12949.937} C_VEL
LIN {X 0,Y 362.162,Z 67.37,A -85,B 0,C 180,E1 -12953.314,E2 -12953.314} C_VEL
LIN {X 0,Y 362.283,Z 67.359,A -85,B 0,C 180,E1 -12957.777,E2 -12957.777} C_VEL
LIN {X 0,Y 362.431,Z 67.34,A -85,B 0,C 180,E1 -12960,E2 -12960} C_VEL
LIN {X 0,Y 362.285,Z 67.356,A -85,B 0,C 180,E1 -12962.224,E2 -12962.224} C_VEL
LIN {X 0,Y 362.129,Z 67.373,A -85,B 0,C 180,E1 -12966.687,E2 -12966.687} C_VEL
LIN {X 0,Y 362.005,Z 67.39,A -85,B 0,C 180,E1 -12970.063,E2 -12970.063} C_VEL
LIN {X 0,Y 362.002,Z 67.39,A -85,B 0,C 180,E1 -12973.899,E2 -12973.899} C_VEL
LIN {X 0,Y 361.932,Z 67.401,A -85,B 0,C 180,E1 -12976.934,E2 -12976.934} C_VEL
LIN {X 0,Y 361.891,Z 67.404,A -85,B 0,C 180,E1 -12980.461,E2 -12980.461} C_VEL
LIN {X 0,Y 361.897,Z 67.402,A -85,B 0,C 180,E1 -12984.113,E2 -12984.113} C_VEL
LIN {X 0,Y 361.868,Z 67.406,A -85,B 0,C 180,E1 -12987.783,E2 -12987.783} C_VEL
LIN {X 0,Y 361.85,Z 67.409,A -85,B 0,C 180,E1 -12991.285,E2 -12991.285} C_VEL
LIN {X 0,Y 361.858,Z 67.41,A -85,B 0,C 180,E1 -12994.28,E2 -12994.28} C_VEL
LIN {X 0,Y 361.866,Z 67.407,A -85,B 0,C 180,E1 -12997.223,E2 -12997.223} C_VEL
LIN {X 0,Y 361.839,Z 67.412,A -85,B 0,C 180,E1 -13000.755,E2 -13000.755} C_VEL
LIN {X 0,Y 361.821,Z 67.417,A -85,B 0,C 180,E1 -13004.368,E2 -13004.368} C_VEL
LIN {X 0,Y 361.835,Z 67.411,A -85,B 0,C 180,E1 -13007.569,E2 -13007.569} C_VEL
LIN {X 0,Y 361.833,Z 67.41,A -85,B 0,C 180,E1 -13010.981,E2 -13010.981} C_VEL
LIN {X 0,Y 361.877,Z 67.405,A -85,B 0,C 180,E1 -13014.655,E2 -13014.655} C_VEL
LIN {X 0,Y 361.84,Z 67.41,A -85,B 0,C 180,E1 -13018.37,E2 -13018.37} C_VEL
LIN {X 0,Y 361.922,Z 67.486,A -85,B 0,C 180,E1 -13020.084,E2 -13020.084} C_VEL
LIN {X 0,Y 364.606,Z 80.214,A -85,B 0,C 180,E1 -13023.076,E2 -13023.076} C_VEL
LIN {X 0,Y 365.262,Z 84.609,A -85,B 0,C 180,E1 -13024.071,E2 -13024.071} C_VEL
LIN {X 0,Y 364.163,Z 98.407,A -85,B 0,C 180,E1 -13026.995,E2 -13026.995} C_VEL
LIN {X 0,Y 363.499,Z 107.351,A -85,B 0,C 180,E1 -13028.861,E2 -13028.861} C_VEL
LIN {X 0,Y 368.148,Z 144.631,A -85,B 0,C 180,E1 -13029.837,E2 -13029.837} C_VEL
LIN {X 0,Y 367.14,Z 216.604,A -85,B 0,C 180,E1 -13031.262,E2 -13031.262} C_VEL
LIN {X 0,Y 366.532,Z 230.561,A -85,B 0,C 180,E1 -13031.773,E2 -13031.773} C_VEL
LIN {X 0,Y 365.691,Z 243.035,A -85,B 0,C 180,E1 -13032.453,E2 -13032.453} C_VEL
LIN {X 0,Y 364.726,Z 254.975,A -85,B 0,C 180,E1 -13033.343,E2 -13033.343} C_VEL
LIN {X 0,Y 363.796,Z 266.471,A -85,B 0,C 180,E1 -13034.452,E2 -13034.452} C_VEL
LIN {X 0,Y 362.84,Z 276.976,A -85,B 0,C 180,E1 -13035.724,E2 -13035.724} C_VEL
LIN {X 0,Y 362.082,Z 286.113,A -85,B 0,C 180,E1 -13037.102,E2 -13037.102} C_VEL
LIN {X 0,Y 361.481,Z 293.782,A -85,B 0,C 180,E1 -13038.505,E2 -13038.505} C_VEL
LIN {X 0,Y 360.918,Z 301.293,A -85,B 0,C 180,E1 -13040.19,E2 -13040.19} C_VEL
LIN {X 0,Y 360.58,Z 308.207,A -85,B 0,C 180,E1 -13042.158,E2 -13042.158} C_VEL
LIN {X 0,Y 360.379,Z 313.187,A -85,B 0,C 180,E1 -13044.038,E2 -13044.038} C_VEL
LIN {X 0,Y 360.472,Z 316.201,A -85,B 0,C 180,E1 -13045.527,E2 -13045.527} C_VEL
LIN {X 0,Y 360.515,Z 319.203,A -85,B 0,C 180,E1 -13047.765,E2 -13047.765} C_VEL
LIN {X 0,Y 360.539,Z 320.097,A -85,B 0,C 180,E1 -13048.883,E2 -13048.883} C_VEL
LIN {X 0,Y 360.521,Z 320.56,A -85,B 0,C 180,E1 -13050,E2 -13050} C_VEL
LIN {X 0,Y 360.518,Z 320.607,A -85,B 0,C 180,E1 -13051.117,E2 -13051.117} C_VEL
